KUKA KRL program: firepit2_1.src

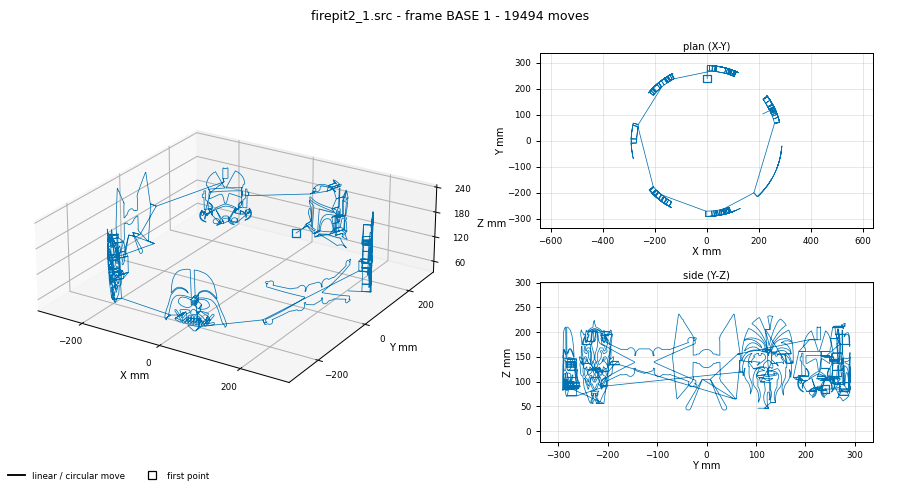
[picture p0: tool path of firepit2_1.src in frame BASE 1, 19494 of 19496 moves have a stored position in this frame; points joined in program order, loops and branches not executed]
&ACCESS RVP
&REL 1
&PARAM TEMPLATE = C:\KRC\Roboter\Template\vorgabe
&PARAM EDITMASK = *
DEF firepit2_1( )
EXT BAS (BAS_COMMAND :IN,REAL :IN )
DECL EKI_STATUS RET

INT INDX
FOR INDX=1 TO 6
	$ACC_AXIS[INDX]=50
	$VEL_AXIS[INDX]=20
ENDFOR

$VEL.ORI1=200
$VEL.ORI2=200
$ACC.ORI1=100
$ACC.ORI2=100

$VEL.CP = 0.1

$ACC.CP = 1

$IPO_MODE = #TCP
$APO.CDIS = 0.5
$ADVANCE = 5

$ACT_TOOL = 1
$TOOL=TOOL_DATA[1]
$ACT_BASE = 1
$BASE=BASE_DATA[1]

RET=EKI_Init("oxy")
RET=EKI_Open("oxy")

RET=EKI_SetBool("oxy","torchState",FALSE)
RET = EKI_Send("oxy","torchState")
PTP {A1 0.0,A2 -100.0,A3 150.0,A4 0.0,A5 -50.0,A6 0.0}

LIN {X 2.269,Y 239.989,Z 85.092,A -90.542,B 90.000,C 0.000} C_DIS
LIN {X 2.723,Y 287.987,Z 85.092,A -90.542,B 90.000,C 0.000} C_DIS
LIN {X 2.742,Y 289.987,Z 85.092,A -90.542,B 90.000,C 0.000} C_DIS
WAIT SEC 1
RET=EKI_SetBool("oxy","torchState",TRUE)
RET = EKI_Send("oxy","torchState")
LIN {X 3.106,Y 289.983,Z 85.575,A -90.614,B 90.000,C 0.000} C_DIS
LIN {X 4.946,Y 289.953,Z 87.268,A -90.977,B 90.000,C 0.000} C_DIS
LIN {X 6.840,Y 289.911,Z 88.899,A -91.352,B 90.000,C 0.000} C_DIS
LIN {X 8.695,Y 289.870,Z 90.495,A -91.718,B 90.000,C 0.000} C_DIS
LIN {X 10.282,Y 289.814,Z 88.565,A -92.032,B 90.000,C 0.000} C_DIS
LIN {X 11.858,Y 289.753,Z 86.625,A -92.343,B 90.000,C 0.000} C_DIS
LIN {X 13.089,Y 289.704,Z 85.109,A -92.587,B 90.000,C 0.000} C_DIS
LIN {X 13.703,Y 289.676,Z 84.499,A -92.708,B 90.000,C 0.000} C_DIS
LIN {X 13.987,Y 289.663,Z 84.366,A -92.764,B 90.000,C 0.000} C_DIS
LIN {X 14.006,Y 289.662,Z 86.866,A -92.768,B 90.000,C 0.000} C_DIS
LIN {X 14.025,Y 289.661,Z 89.365,A -92.772,B 90.000,C 0.000} C_DIS
LIN {X 14.045,Y 289.660,Z 91.865,A -92.776,B 90.000,C 0.000} C_DIS
LIN {X 14.064,Y 289.659,Z 94.365,A -92.780,B 90.000,C 0.000} C_DIS
LIN {X 14.084,Y 289.658,Z 96.865,A -92.784,B 90.000,C 0.000} C_DIS
LIN {X 14.103,Y 289.657,Z 99.365,A -92.788,B 90.000,C 0.000} C_DIS
LIN {X 14.116,Y 289.656,Z 101.865,A -92.790,B 90.000,C 0.000} C_DIS
LIN {X 14.110,Y 289.657,Z 104.365,A -92.789,B 90.000,C 0.000} C_DIS
LIN {X 14.104,Y 289.657,Z 106.864,A -92.788,B 90.000,C 0.000} C_DIS
LIN {X 14.098,Y 289.657,Z 109.364,A -92.786,B 90.000,C 0.000} C_DIS
LIN {X 14.092,Y 289.657,Z 111.864,A -92.785,B 90.000,C 0.000} C_DIS
LIN {X 14.086,Y 289.658,Z 114.364,A -92.784,B 90.000,C 0.000} C_DIS
LIN {X 14.080,Y 289.658,Z 116.864,A -92.783,B 90.000,C 0.000} C_DIS
LIN {X 14.074,Y 289.658,Z 119.364,A -92.782,B 90.000,C 0.000} C_DIS
LIN {X 13.921,Y 289.666,Z 121.859,A -92.751,B 90.000,C 0.000} C_DIS
LIN {X 13.726,Y 289.675,Z 124.352,A -92.713,B 90.000,C 0.000} C_DIS
LIN {X 13.394,Y 289.691,Z 126.829,A -92.647,B 90.000,C 0.000} C_DIS
LIN {X 12.905,Y 289.713,Z 129.281,A -92.550,B 90.000,C 0.000} C_DIS
LIN {X 12.266,Y 289.740,Z 131.697,A -92.424,B 90.000,C 0.000} C_DIS
LIN {X 11.477,Y 289.773,Z 134.069,A -92.268,B 90.000,C 0.000} C_DIS
LIN {X 10.547,Y 289.808,Z 136.390,A -92.084,B 90.000,C 0.000} C_DIS
LIN {X 9.438,Y 289.844,Z 138.630,A -91.865,B 90.000,C 0.000} C_DIS
LIN {X 8.303,Y 289.880,Z 140.857,A -91.641,B 90.000,C 0.000} C_DIS
LIN {X 7.391,Y 289.906,Z 142.534,A -91.460,B 90.000,C 0.000} C_DIS
LIN {X 7.419,Y 289.905,Z 145.034,A -91.466,B 90.000,C 0.000} C_DIS
LIN {X 7.484,Y 289.903,Z 147.533,A -91.479,B 90.000,C 0.000} C_DIS
LIN {X 7.552,Y 289.902,Z 149.639,A -91.492,B 90.000,C 0.000} C_DIS
LIN {X 7.695,Y 289.898,Z 150.255,A -91.521,B 90.000,C 0.000} C_DIS
LIN {X 7.879,Y 289.893,Z 150.291,A -91.557,B 90.000,C 0.000} C_DIS
LIN {X 8.002,Y 289.890,Z 150.193,A -91.581,B 90.000,C 0.000} C_DIS
LIN {X 8.394,Y 289.878,Z 148.728,A -91.659,B 90.000,C 0.000} C_DIS
LIN {X 8.824,Y 289.866,Z 147.667,A -91.744,B 90.000,C 0.000} C_DIS
LIN {X 9.375,Y 289.848,Z 146.647,A -91.853,B 90.000,C 0.000} C_DIS
LIN {X 10.028,Y 289.827,Z 145.711,A -91.982,B 90.000,C 0.000} C_DIS
LIN {X 11.083,Y 289.788,Z 144.578,A -92.190,B 90.000,C 0.000} C_DIS
LIN {X 13.041,Y 289.706,Z 143.026,A -92.577,B 90.000,C 0.000} C_DIS
LIN {X 15.151,Y 289.602,Z 141.689,A -92.995,B 90.000,C 0.000} C_DIS
LIN {X 17.324,Y 289.482,Z 140.459,A -93.425,B 90.000,C 0.000} C_DIS
LIN {X 17.924,Y 289.446,Z 140.050,A -93.544,B 90.000,C 0.000} C_DIS
LIN {X 18.369,Y 289.418,Z 139.616,A -93.632,B 90.000,C 0.000} C_DIS
LIN {X 18.808,Y 289.389,Z 139.037,A -93.719,B 90.000,C 0.000} C_DIS
LIN {X 19.190,Y 289.364,Z 138.387,A -93.794,B 90.000,C 0.000} C_DIS
LIN {X 19.466,Y 289.346,Z 137.743,A -93.849,B 90.000,C 0.000} C_DIS
LIN {X 19.578,Y 289.338,Z 137.136,A -93.871,B 90.000,C 0.000} C_DIS
LIN {X 19.405,Y 289.350,Z 134.642,A -93.837,B 90.000,C 0.000} C_DIS
LIN {X 19.241,Y 289.361,Z 132.148,A -93.804,B 90.000,C 0.000} C_DIS
LIN {X 19.076,Y 289.372,Z 129.653,A -93.772,B 90.000,C 0.000} C_DIS
LIN {X 18.917,Y 289.382,Z 127.158,A -93.740,B 90.000,C 0.000} C_DIS
LIN {X 18.761,Y 289.391,Z 124.663,A -93.709,B 90.000,C 0.000} C_DIS
LIN {X 18.606,Y 289.401,Z 122.168,A -93.678,B 90.000,C 0.000} C_DIS
LIN {X 18.450,Y 289.410,Z 119.673,A -93.648,B 90.000,C 0.000} C_DIS
LIN {X 18.294,Y 289.420,Z 117.178,A -93.617,B 90.000,C 0.000} C_DIS
LIN {X 18.138,Y 289.429,Z 114.683,A -93.586,B 90.000,C 0.000} C_DIS
LIN {X 17.983,Y 289.439,Z 112.188,A -93.555,B 90.000,C 0.000} C_DIS
LIN {X 17.827,Y 289.448,Z 109.693,A -93.524,B 90.000,C 0.000} C_DIS
LIN {X 17.671,Y 289.458,Z 107.198,A -93.493,B 90.000,C 0.000} C_DIS
LIN {X 17.515,Y 289.467,Z 104.703,A -93.463,B 90.000,C 0.000} C_DIS
LIN {X 17.359,Y 289.477,Z 102.208,A -93.432,B 90.000,C 0.000} C_DIS
LIN {X 17.204,Y 289.486,Z 99.713,A -93.401,B 90.000,C 0.000} C_DIS
LIN {X 17.048,Y 289.496,Z 97.218,A -93.370,B 90.000,C 0.000} C_DIS
LIN {X 16.892,Y 289.505,Z 94.723,A -93.339,B 90.000,C 0.000} C_DIS
LIN {X 16.736,Y 289.515,Z 92.228,A -93.308,B 90.000,C 0.000} C_DIS
LIN {X 16.580,Y 289.524,Z 89.733,A -93.278,B 90.000,C 0.000} C_DIS
LIN {X 16.425,Y 289.534,Z 87.238,A -93.247,B 90.000,C 0.000} C_DIS
LIN {X 16.269,Y 289.543,Z 84.743,A -93.216,B 90.000,C 0.000} C_DIS
LIN {X 16.179,Y 289.548,Z 83.458,A -93.198,B 90.000,C 0.000} C_DIS
LIN {X 18.542,Y 289.403,Z 82.655,A -93.666,B 90.000,C 0.000} C_DIS
LIN {X 20.897,Y 289.243,Z 81.832,A -94.132,B 90.000,C 0.000} C_DIS
LIN {X 23.250,Y 289.066,Z 81.005,A -94.598,B 90.000,C 0.000} C_DIS
LIN {X 24.631,Y 288.952,Z 80.507,A -94.872,B 90.000,C 0.000} C_DIS
LIN {X 23.274,Y 289.064,Z 78.411,A -94.603,B 90.000,C 0.000} C_DIS
LIN {X 21.895,Y 289.172,Z 76.398,A -94.330,B 90.000,C 0.000} C_DIS
LIN {X 19.621,Y 289.332,Z 77.424,A -93.880,B 90.000,C 0.000} C_DIS
LIN {X 17.348,Y 289.477,Z 78.455,A -93.430,B 90.000,C 0.000} C_DIS
LIN {X 15.074,Y 289.606,Z 79.486,A -92.980,B 90.000,C 0.000} C_DIS
LIN {X 12.800,Y 289.716,Z 80.517,A -92.530,B 90.000,C 0.000} C_DIS
LIN {X 10.524,Y 289.807,Z 81.548,A -92.080,B 90.000,C 0.000} C_DIS
LIN {X 8.248,Y 289.880,Z 82.580,A -91.630,B 90.000,C 0.000} C_DIS
LIN {X 5.972,Y 289.936,Z 83.611,A -91.180,B 90.000,C 0.000} C_DIS
LIN {X 3.698,Y 289.975,Z 84.650,A -90.731,B 90.000,C 0.000} C_DIS
LIN {X 2.742,Y 289.987,Z 85.092,A -90.542,B 90.000,C 0.000} C_DIS
LIN {X 2.723,Y 287.987,Z 85.092,A -90.542,B 90.000,C 0.000} C_DIS
WAIT SEC 0.1
RET=EKI_SetBool("oxy","torchState",FALSE)
RET = EKI_Send("oxy","torchState")
LIN {X 2.553,Y 269.988,Z 85.092,A -90.542,B 90.000,C 0.000} C_DIS
LIN {X 10.715,Y 269.787,Z 97.827,A -92.274,B 90.000,C 0.000} C_DIS
LIN {X 11.429,Y 287.773,Z 97.827,A -92.274,B 90.000,C 0.000} C_DIS
LIN {X 11.508,Y 289.772,Z 97.827,A -92.274,B 90.000,C 0.000} C_DIS
WAIT SEC 1
RET=EKI_SetBool("oxy","torchState",TRUE)
RET = EKI_Send("oxy","torchState")
LIN {X 11.733,Y 289.763,Z 98.367,A -92.319,B 90.000,C 0.000} C_DIS
LIN {X 12.293,Y 289.739,Z 100.803,A -92.430,B 90.000,C 0.000} C_DIS
LIN {X 12.626,Y 289.725,Z 103.281,A -92.495,B 90.000,C 0.000} C_DIS
LIN {X 12.812,Y 289.717,Z 105.774,A -92.532,B 90.000,C 0.000} C_DIS
LIN {X 12.854,Y 289.715,Z 108.274,A -92.540,B 90.000,C 0.000} C_DIS
LIN {X 12.814,Y 289.717,Z 110.773,A -92.533,B 90.000,C 0.000} C_DIS
LIN {X 12.625,Y 289.725,Z 113.266,A -92.495,B 90.000,C 0.000} C_DIS
LIN {X 12.426,Y 289.734,Z 115.758,A -92.456,B 90.000,C 0.000} C_DIS
LIN {X 12.102,Y 289.747,Z 118.237,A -92.392,B 90.000,C 0.000} C_DIS
LIN {X 11.760,Y 289.761,Z 120.713,A -92.324,B 90.000,C 0.000} C_DIS
LIN {X 11.291,Y 289.780,Z 123.169,A -92.231,B 90.000,C 0.000} C_DIS
LIN {X 10.772,Y 289.800,Z 125.614,A -92.129,B 90.000,C 0.000} C_DIS
LIN {X 10.082,Y 289.825,Z 128.017,A -91.992,B 90.000,C 0.000} C_DIS
LIN {X 9.685,Y 289.838,Z 128.998,A -91.914,B 90.000,C 0.000} C_DIS
LIN {X 9.310,Y 289.851,Z 129.580,A -91.840,B 90.000,C 0.000} C_DIS
LIN {X 8.906,Y 289.863,Z 129.935,A -91.760,B 90.000,C 0.000} C_DIS
LIN {X 8.480,Y 289.876,Z 130.055,A -91.676,B 90.000,C 0.000} C_DIS
LIN {X 8.053,Y 289.888,Z 129.956,A -91.591,B 90.000,C 0.000} C_DIS
LIN {X 7.635,Y 289.899,Z 129.594,A -91.509,B 90.000,C 0.000} C_DIS
LIN {X 7.309,Y 289.908,Z 129.126,A -91.444,B 90.000,C 0.000} C_DIS
LIN {X 6.981,Y 289.916,Z 128.453,A -91.379,B 90.000,C 0.000} C_DIS
LIN {X 6.222,Y 289.933,Z 126.072,A -91.229,B 90.000,C 0.000} C_DIS
LIN {X 5.689,Y 289.944,Z 123.629,A -91.124,B 90.000,C 0.000} C_DIS
LIN {X 5.315,Y 289.951,Z 121.157,A -91.050,B 90.000,C 0.000} C_DIS
LIN {X 5.080,Y 289.955,Z 118.668,A -91.004,B 90.000,C 0.000} C_DIS
LIN {X 4.862,Y 289.959,Z 116.354,A -90.961,B 90.000,C 0.000} C_DIS
LIN {X 4.950,Y 289.958,Z 115.800,A -90.978,B 90.000,C 0.000} C_DIS
LIN {X 6.205,Y 289.933,Z 113.638,A -91.226,B 90.000,C 0.000} C_DIS
LIN {X 6.480,Y 289.928,Z 113.155,A -91.280,B 90.000,C 0.000} C_DIS
LIN {X 7.462,Y 289.904,Z 110.856,A -91.474,B 90.000,C 0.000} C_DIS
LIN {X 8.309,Y 289.880,Z 108.504,A -91.642,B 90.000,C 0.000} C_DIS
LIN {X 9.087,Y 289.857,Z 106.128,A -91.796,B 90.000,C 0.000} C_DIS
LIN {X 9.799,Y 289.834,Z 103.732,A -91.936,B 90.000,C 0.000} C_DIS
LIN {X 10.498,Y 289.809,Z 101.332,A -92.075,B 90.000,C 0.000} C_DIS
LIN {X 11.191,Y 289.783,Z 98.930,A -92.211,B 90.000,C 0.000} C_DIS
LIN {X 11.508,Y 289.772,Z 97.827,A -92.274,B 90.000,C 0.000} C_DIS
LIN {X 11.429,Y 287.773,Z 97.827,A -92.274,B 90.000,C 0.000} C_DIS
WAIT SEC 0.1
RET=EKI_SetBool("oxy","torchState",FALSE)
RET = EKI_Send("oxy","torchState")
LIN {X 10.715,Y 269.787,Z 97.827,A -92.274,B 90.000,C 0.000} C_DIS
LIN {X 30.888,Y 268.227,Z 79.694,A -96.569,B 90.000,C 0.000} C_DIS
LIN {X 32.947,Y 286.109,Z 79.694,A -96.569,B 90.000,C 0.000} C_DIS
LIN {X 33.176,Y 288.096,Z 79.694,A -96.569,B 90.000,C 0.000} C_DIS
WAIT SEC 1
RET=EKI_SetBool("oxy","torchState",TRUE)
RET = EKI_Send("oxy","torchState")
LIN {X 31.366,Y 288.299,Z 79.726,A -96.209,B 90.000,C 0.000} C_DIS
LIN {X 31.245,Y 288.312,Z 79.795,A -96.185,B 90.000,C 0.000} C_DIS
LIN {X 31.374,Y 288.298,Z 82.291,A -96.211,B 90.000,C 0.000} C_DIS
LIN {X 31.521,Y 288.282,Z 84.787,A -96.240,B 90.000,C 0.000} C_DIS
LIN {X 31.668,Y 288.266,Z 87.283,A -96.269,B 90.000,C 0.000} C_DIS
LIN {X 31.819,Y 288.249,Z 89.778,A -96.299,B 90.000,C 0.000} C_DIS
LIN {X 31.971,Y 288.232,Z 92.273,A -96.329,B 90.000,C 0.000} C_DIS
LIN {X 32.123,Y 288.215,Z 94.768,A -96.360,B 90.000,C 0.000} C_DIS
LIN {X 32.275,Y 288.198,Z 97.264,A -96.390,B 90.000,C 0.000} C_DIS
LIN {X 32.427,Y 288.181,Z 99.759,A -96.420,B 90.000,C 0.000} C_DIS
LIN {X 32.579,Y 288.164,Z 102.254,A -96.450,B 90.000,C 0.000} C_DIS
LIN {X 32.731,Y 288.147,Z 104.749,A -96.481,B 90.000,C 0.000} C_DIS
LIN {X 32.878,Y 288.130,Z 107.245,A -96.510,B 90.000,C 0.000} C_DIS
LIN {X 33.024,Y 288.114,Z 109.741,A -96.539,B 90.000,C 0.000} C_DIS
LIN {X 33.165,Y 288.097,Z 112.236,A -96.567,B 90.000,C 0.000} C_DIS
LIN {X 33.305,Y 288.081,Z 114.732,A -96.595,B 90.000,C 0.000} C_DIS
LIN {X 33.446,Y 288.065,Z 117.228,A -96.623,B 90.000,C 0.000} C_DIS
LIN {X 33.590,Y 288.048,Z 119.724,A -96.651,B 90.000,C 0.000} C_DIS
LIN {X 33.747,Y 288.030,Z 122.219,A -96.683,B 90.000,C 0.000} C_DIS
LIN {X 33.904,Y 288.011,Z 124.714,A -96.714,B 90.000,C 0.000} C_DIS
LIN {X 34.055,Y 287.993,Z 127.209,A -96.744,B 90.000,C 0.000} C_DIS
LIN {X 34.202,Y 287.976,Z 129.705,A -96.773,B 90.000,C 0.000} C_DIS
LIN {X 34.346,Y 287.959,Z 132.200,A -96.802,B 90.000,C 0.000} C_DIS
LIN {X 34.409,Y 287.951,Z 133.346,A -96.814,B 90.000,C 0.000} C_DIS
LIN {X 34.518,Y 287.938,Z 133.760,A -96.836,B 90.000,C 0.000} C_DIS
LIN {X 34.705,Y 287.916,Z 134.075,A -96.873,B 90.000,C 0.000} C_DIS
LIN {X 34.992,Y 287.881,Z 134.376,A -96.930,B 90.000,C 0.000} C_DIS
LIN {X 35.373,Y 287.835,Z 134.609,A -97.006,B 90.000,C 0.000} C_DIS
LIN {X 36.438,Y 287.702,Z 134.880,A -97.218,B 90.000,C 0.000} C_DIS
LIN {X 38.916,Y 287.375,Z 134.943,A -97.712,B 90.000,C 0.000} C_DIS
LIN {X 41.391,Y 287.029,Z 134.988,A -98.206,B 90.000,C 0.000} C_DIS
LIN {X 43.863,Y 286.659,Z 135.032,A -98.700,B 90.000,C 0.000} C_DIS
LIN {X 46.332,Y 286.270,Z 135.076,A -99.193,B 90.000,C 0.000} C_DIS
LIN {X 48.798,Y 285.862,Z 135.148,A -99.687,B 90.000,C 0.000} C_DIS
LIN {X 51.256,Y 285.434,Z 135.304,A -100.180,B 90.000,C 0.000} C_DIS
LIN {X 53.709,Y 284.981,Z 135.460,A -100.673,B 90.000,C 0.000} C_DIS
LIN {X 56.159,Y 284.507,Z 135.616,A -101.166,B 90.000,C 0.000} C_DIS
LIN {X 58.601,Y 284.010,Z 135.814,A -101.658,B 90.000,C 0.000} C_DIS
LIN {X 61.038,Y 283.501,Z 136.040,A -102.150,B 90.000,C 0.000} C_DIS
LIN {X 63.463,Y 282.964,Z 136.326,A -102.641,B 90.000,C 0.000} C_DIS
LIN {X 65.880,Y 282.414,Z 136.644,A -103.131,B 90.000,C 0.000} C_DIS
LIN {X 68.285,Y 281.844,Z 137.022,A -103.619,B 90.000,C 0.000} C_DIS
LIN {X 70.670,Y 281.253,Z 137.484,A -104.105,B 90.000,C 0.000} C_DIS
LIN {X 73.034,Y 280.648,Z 138.026,A -104.587,B 90.000,C 0.000} C_DIS
LIN {X 75.378,Y 280.032,Z 138.640,A -105.066,B 90.000,C 0.000} C_DIS
LIN {X 76.863,Y 279.629,Z 139.139,A -105.370,B 90.000,C 0.000} C_DIS
LIN {X 76.918,Y 279.613,Z 139.927,A -105.381,B 90.000,C 0.000} C_DIS
LIN {X 76.873,Y 279.626,Z 140.646,A -105.372,B 90.000,C 0.000} C_DIS
LIN {X 74.460,Y 280.277,Z 140.616,A -104.878,B 90.000,C 0.000} C_DIS
LIN {X 72.040,Y 280.907,Z 140.607,A -104.384,B 90.000,C 0.000} C_DIS
LIN {X 69.616,Y 281.516,Z 140.598,A -103.890,B 90.000,C 0.000} C_DIS
LIN {X 67.186,Y 282.106,Z 140.611,A -103.396,B 90.000,C 0.000} C_DIS
LIN {X 64.753,Y 282.676,Z 140.646,A -102.902,B 90.000,C 0.000} C_DIS
LIN {X 62.314,Y 283.226,Z 140.681,A -102.408,B 90.000,C 0.000} C_DIS
LIN {X 59.872,Y 283.749,Z 140.789,A -101.915,B 90.000,C 0.000} C_DIS
LIN {X 57.426,Y 284.253,Z 140.900,A -101.421,B 90.000,C 0.000} C_DIS
LIN {X 54.977,Y 284.737,Z 141.035,A -100.928,B 90.000,C 0.000} C_DIS
LIN {X 52.526,Y 285.200,Z 141.195,A -100.435,B 90.000,C 0.000} C_DIS
LIN {X 50.071,Y 285.643,Z 141.363,A -99.942,B 90.000,C 0.000} C_DIS
LIN {X 47.616,Y 286.064,Z 141.575,A -99.450,B 90.000,C 0.000} C_DIS
LIN {X 45.157,Y 286.461,Z 141.787,A -98.958,B 90.000,C 0.000} C_DIS
LIN {X 42.699,Y 286.837,Z 142.045,A -98.467,B 90.000,C 0.000} C_DIS
LIN {X 40.238,Y 287.192,Z 142.311,A -97.976,B 90.000,C 0.000} C_DIS
LIN {X 37.779,Y 287.521,Z 142.611,A -97.485,B 90.000,C 0.000} C_DIS
LIN {X 35.320,Y 287.838,Z 142.936,A -96.996,B 90.000,C 0.000} C_DIS
LIN {X 32.867,Y 288.124,Z 143.323,A -96.508,B 90.000,C 0.000} C_DIS
LIN {X 30.417,Y 288.398,Z 143.738,A -96.021,B 90.000,C 0.000} C_DIS
LIN {X 27.978,Y 288.642,Z 144.228,A -95.536,B 90.000,C 0.000} C_DIS
LIN {X 25.548,Y 288.867,Z 144.773,A -95.054,B 90.000,C 0.000} C_DIS
LIN {X 23.128,Y 289.075,Z 145.363,A -94.574,B 90.000,C 0.000} C_DIS
LIN {X 20.731,Y 289.253,Z 146.048,A -94.099,B 90.000,C 0.000} C_DIS
LIN {X 18.356,Y 289.415,Z 146.813,A -93.629,B 90.000,C 0.000} C_DIS
LIN {X 16.021,Y 289.555,Z 147.694,A -93.167,B 90.000,C 0.000} C_DIS
LIN {X 14.146,Y 289.655,Z 148.532,A -92.796,B 90.000,C 0.000} C_DIS
LIN {X 12.056,Y 289.749,Z 149.750,A -92.383,B 90.000,C 0.000} C_DIS
LIN {X 10.680,Y 289.803,Z 150.791,A -92.110,B 90.000,C 0.000} C_DIS
LIN {X 9.525,Y 289.844,Z 151.907,A -91.882,B 90.000,C 0.000} C_DIS
LIN {X 8.647,Y 289.871,Z 153.037,A -91.709,B 90.000,C 0.000} C_DIS
LIN {X 8.100,Y 289.887,Z 154.122,A -91.601,B 90.000,C 0.000} C_DIS
LIN {X 7.966,Y 289.891,Z 154.614,A -91.574,B 90.000,C 0.000} C_DIS
LIN {X 7.936,Y 289.891,Z 155.165,A -91.568,B 90.000,C 0.000} C_DIS
LIN {X 8.018,Y 289.889,Z 156.091,A -91.584,B 90.000,C 0.000} C_DIS
LIN {X 8.873,Y 289.864,Z 158.440,A -91.753,B 90.000,C 0.000} C_DIS
LIN {X 9.052,Y 289.859,Z 158.884,A -91.789,B 90.000,C 0.000} C_DIS
LIN {X 11.147,Y 289.779,Z 157.522,A -92.203,B 90.000,C 0.000} C_DIS
LIN {X 13.204,Y 289.689,Z 156.104,A -92.610,B 90.000,C 0.000} C_DIS
LIN {X 15.264,Y 289.598,Z 154.691,A -93.017,B 90.000,C 0.000} C_DIS
LIN {X 17.393,Y 289.476,Z 153.386,A -93.438,B 90.000,C 0.000} C_DIS
LIN {X 19.610,Y 289.333,Z 152.240,A -93.877,B 90.000,C 0.000} C_DIS
LIN {X 21.892,Y 289.170,Z 151.232,A -94.329,B 90.000,C 0.000} C_DIS
LIN {X 24.232,Y 288.984,Z 150.371,A -94.793,B 90.000,C 0.000} C_DIS
LIN {X 26.612,Y 288.774,Z 149.635,A -95.265,B 90.000,C 0.000} C_DIS
LIN {X 29.022,Y 288.541,Z 149.013,A -95.744,B 90.000,C 0.000} C_DIS
LIN {X 31.454,Y 288.286,Z 148.495,A -96.227,B 90.000,C 0.000} C_DIS
LIN {X 33.902,Y 288.008,Z 148.069,A -96.713,B 90.000,C 0.000} C_DIS
LIN {X 36.360,Y 287.709,Z 147.727,A -97.203,B 90.000,C 0.000} C_DIS
LIN {X 38.825,Y 287.389,Z 147.457,A -97.694,B 90.000,C 0.000} C_DIS
LIN {X 41.293,Y 287.043,Z 147.270,A -98.186,B 90.000,C 0.000} C_DIS
LIN {X 43.763,Y 286.676,Z 147.143,A -98.680,B 90.000,C 0.000} C_DIS
LIN {X 46.230,Y 286.288,Z 147.033,A -99.173,B 90.000,C 0.000} C_DIS
LIN {X 48.694,Y 285.879,Z 146.923,A -99.666,B 90.000,C 0.000} C_DIS
LIN {X 51.155,Y 285.450,Z 146.840,A -100.160,B 90.000,C 0.000} C_DIS
LIN {X 53.614,Y 284.998,Z 146.795,A -100.654,B 90.000,C 0.000} C_DIS
LIN {X 56.068,Y 284.526,Z 146.750,A -101.148,B 90.000,C 0.000} C_DIS
LIN {X 58.519,Y 284.032,Z 146.727,A -101.642,B 90.000,C 0.000} C_DIS
LIN {X 60.965,Y 283.518,Z 146.769,A -102.136,B 90.000,C 0.000} C_DIS
LIN {X 63.406,Y 282.983,Z 146.811,A -102.629,B 90.000,C 0.000} C_DIS
LIN {X 65.843,Y 282.425,Z 146.853,A -103.123,B 90.000,C 0.000} C_DIS
LIN {X 68.274,Y 281.847,Z 146.940,A -103.617,B 90.000,C 0.000} C_DIS
LIN {X 70.699,Y 281.249,Z 147.031,A -104.110,B 90.000,C 0.000} C_DIS
LIN {X 73.119,Y 280.629,Z 147.122,A -104.604,B 90.000,C 0.000} C_DIS
LIN {X 75.532,Y 279.983,Z 147.233,A -105.097,B 90.000,C 0.000} C_DIS
LIN {X 77.942,Y 279.329,Z 147.350,A -105.591,B 90.000,C 0.000} C_DIS
LIN {X 80.341,Y 278.640,Z 147.491,A -106.084,B 90.000,C 0.000} C_DIS
LIN {X 82.738,Y 277.946,Z 147.637,A -106.577,B 90.000,C 0.000} C_DIS
LIN {X 83.639,Y 277.677,Z 147.701,A -106.763,B 90.000,C 0.000} C_DIS
LIN {X 84.426,Y 277.439,Z 147.637,A -106.925,B 90.000,C 0.000} C_DIS
LIN {X 85.212,Y 277.198,Z 146.852,A -107.088,B 90.000,C 0.000} C_DIS
LIN {X 85.569,Y 277.088,Z 146.663,A -107.161,B 90.000,C 0.000} C_DIS
LIN {X 85.692,Y 277.050,Z 146.577,A -107.187,B 90.000,C 0.000} C_DIS
LIN {X 85.754,Y 277.031,Z 146.399,A -107.200,B 90.000,C 0.000} C_DIS
LIN {X 85.652,Y 277.063,Z 143.901,A -107.179,B 90.000,C 0.000} C_DIS
LIN {X 85.533,Y 277.099,Z 141.404,A -107.154,B 90.000,C 0.000} C_DIS
LIN {X 85.455,Y 277.124,Z 138.906,A -107.138,B 90.000,C 0.000} C_DIS
LIN {X 85.383,Y 277.146,Z 136.407,A -107.123,B 90.000,C 0.000} C_DIS
LIN {X 85.314,Y 277.167,Z 133.908,A -107.109,B 90.000,C 0.000} C_DIS
LIN {X 85.248,Y 277.187,Z 131.409,A -107.095,B 90.000,C 0.000} C_DIS
LIN {X 85.166,Y 277.212,Z 128.911,A -107.078,B 90.000,C 0.000} C_DIS
LIN {X 85.080,Y 277.239,Z 126.412,A -107.060,B 90.000,C 0.000} C_DIS
LIN {X 84.986,Y 277.268,Z 123.914,A -107.041,B 90.000,C 0.000} C_DIS
LIN {X 84.904,Y 277.293,Z 121.416,A -107.024,B 90.000,C 0.000} C_DIS
LIN {X 84.828,Y 277.316,Z 118.917,A -107.008,B 90.000,C 0.000} C_DIS
LIN {X 84.756,Y 277.338,Z 116.418,A -106.993,B 90.000,C 0.000} C_DIS
LIN {X 84.678,Y 277.362,Z 113.920,A -106.977,B 90.000,C 0.000} C_DIS
LIN {X 84.595,Y 277.387,Z 111.421,A -106.960,B 90.000,C 0.000} C_DIS
LIN {X 84.513,Y 277.412,Z 108.923,A -106.943,B 90.000,C 0.000} C_DIS
LIN {X 84.431,Y 277.437,Z 106.425,A -106.926,B 90.000,C 0.000} C_DIS
LIN {X 84.352,Y 277.461,Z 103.926,A -106.910,B 90.000,C 0.000} C_DIS
LIN {X 84.259,Y 277.490,Z 101.428,A -106.891,B 90.000,C 0.000} C_DIS
LIN {X 84.162,Y 277.519,Z 98.930,A -106.871,B 90.000,C 0.000} C_DIS
LIN {X 84.095,Y 277.539,Z 96.431,A -106.857,B 90.000,C 0.000} C_DIS
LIN {X 84.031,Y 277.559,Z 93.932,A -106.844,B 90.000,C 0.000} C_DIS
LIN {X 84.008,Y 277.566,Z 93.174,A -106.839,B 90.000,C 0.000} C_DIS
LIN {X 83.913,Y 277.594,Z 92.829,A -106.819,B 90.000,C 0.000} C_DIS
LIN {X 83.739,Y 277.647,Z 92.621,A -106.784,B 90.000,C 0.000} C_DIS
LIN {X 81.633,Y 278.273,Z 91.430,A -106.349,B 90.000,C 0.000} C_DIS
LIN {X 81.536,Y 278.302,Z 91.383,A -106.329,B 90.000,C 0.000} C_DIS
LIN {X 81.573,Y 278.291,Z 93.883,A -106.337,B 90.000,C 0.000} C_DIS
LIN {X 81.610,Y 278.280,Z 96.382,A -106.345,B 90.000,C 0.000} C_DIS
LIN {X 81.647,Y 278.269,Z 98.882,A -106.352,B 90.000,C 0.000} C_DIS
LIN {X 81.683,Y 278.259,Z 101.382,A -106.360,B 90.000,C 0.000} C_DIS
LIN {X 81.726,Y 278.246,Z 103.881,A -106.368,B 90.000,C 0.000} C_DIS
LIN {X 81.770,Y 278.233,Z 106.381,A -106.378,B 90.000,C 0.000} C_DIS
LIN {X 81.814,Y 278.220,Z 108.880,A -106.387,B 90.000,C 0.000} C_DIS
LIN {X 81.858,Y 278.207,Z 111.380,A -106.396,B 90.000,C 0.000} C_DIS
LIN {X 81.903,Y 278.194,Z 113.879,A -106.405,B 90.000,C 0.000} C_DIS
LIN {X 81.947,Y 278.181,Z 116.379,A -106.414,B 90.000,C 0.000} C_DIS
LIN {X 81.987,Y 278.169,Z 118.878,A -106.422,B 90.000,C 0.000} C_DIS
LIN {X 82.025,Y 278.158,Z 121.378,A -106.430,B 90.000,C 0.000} C_DIS
LIN {X 82.063,Y 278.147,Z 123.877,A -106.438,B 90.000,C 0.000} C_DIS
LIN {X 82.105,Y 278.134,Z 126.377,A -106.447,B 90.000,C 0.000} C_DIS
LIN {X 82.119,Y 278.130,Z 128.877,A -106.449,B 90.000,C 0.000} C_DIS
LIN {X 82.056,Y 278.149,Z 130.204,A -106.436,B 90.000,C 0.000} C_DIS
LIN {X 81.775,Y 278.232,Z 130.973,A -106.378,B 90.000,C 0.000} C_DIS
LIN {X 81.315,Y 278.367,Z 131.602,A -106.284,B 90.000,C 0.000} C_DIS
LIN {X 80.724,Y 278.538,Z 132.042,A -106.162,B 90.000,C 0.000} C_DIS
LIN {X 80.050,Y 278.733,Z 132.243,A -106.024,B 90.000,C 0.000} C_DIS
LIN {X 77.654,Y 279.406,Z 132.000,A -105.532,B 90.000,C 0.000} C_DIS
LIN {X 75.264,Y 280.057,Z 131.669,A -105.042,B 90.000,C 0.000} C_DIS
LIN {X 72.870,Y 280.688,Z 131.321,A -104.553,B 90.000,C 0.000} C_DIS
LIN {X 70.480,Y 281.298,Z 130.915,A -104.066,B 90.000,C 0.000} C_DIS
LIN {X 68.094,Y 281.890,Z 130.460,A -103.580,B 90.000,C 0.000} C_DIS
LIN {X 65.716,Y 282.449,Z 129.931,A -103.098,B 90.000,C 0.000} C_DIS
LIN {X 63.344,Y 282.995,Z 129.358,A -102.617,B 90.000,C 0.000} C_DIS
LIN {X 60.991,Y 283.512,Z 128.692,A -102.141,B 90.000,C 0.000} C_DIS
LIN {X 58.675,Y 283.999,Z 127.886,A -101.673,B 90.000,C 0.000} C_DIS
LIN {X 56.409,Y 284.458,Z 126.935,A -101.216,B 90.000,C 0.000} C_DIS
LIN {X 54.210,Y 284.887,Z 125.825,A -100.774,B 90.000,C 0.000} C_DIS
LIN {X 52.122,Y 285.277,Z 124.507,A -100.354,B 90.000,C 0.000} C_DIS
LIN {X 50.180,Y 285.625,Z 122.972,A -99.964,B 90.000,C 0.000} C_DIS
LIN {X 48.375,Y 285.936,Z 121.271,A -99.602,B 90.000,C 0.000} C_DIS
LIN {X 46.695,Y 286.214,Z 119.440,A -99.266,B 90.000,C 0.000} C_DIS
LIN {X 46.031,Y 286.323,Z 118.709,A -99.133,B 90.000,C 0.000} C_DIS
LIN {X 44.565,Y 286.554,Z 116.698,A -98.840,B 90.000,C 0.000} C_DIS
LIN {X 43.228,Y 286.759,Z 114.595,A -98.573,B 90.000,C 0.000} C_DIS
LIN {X 42.019,Y 286.939,Z 112.415,A -98.331,B 90.000,C 0.000} C_DIS
LIN {X 40.925,Y 287.098,Z 110.172,A -98.113,B 90.000,C 0.000} C_DIS
LIN {X 40.001,Y 287.227,Z 107.853,A -97.928,B 90.000,C 0.000} C_DIS
LIN {X 39.171,Y 287.342,Z 105.498,A -97.763,B 90.000,C 0.000} C_DIS
LIN {X 38.415,Y 287.444,Z 103.117,A -97.612,B 90.000,C 0.000} C_DIS
LIN {X 37.801,Y 287.525,Z 100.695,A -97.490,B 90.000,C 0.000} C_DIS
LIN {X 37.242,Y 287.599,Z 98.259,A -97.378,B 90.000,C 0.000} C_DIS
LIN {X 36.760,Y 287.661,Z 95.807,A -97.282,B 90.000,C 0.000} C_DIS
LIN {X 36.360,Y 287.711,Z 93.340,A -97.203,B 90.000,C 0.000} C_DIS
LIN {X 35.997,Y 287.757,Z 90.867,A -97.130,B 90.000,C 0.000} C_DIS
LIN {X 35.724,Y 287.791,Z 88.382,A -97.076,B 90.000,C 0.000} C_DIS
LIN {X 35.466,Y 287.823,Z 85.896,A -97.025,B 90.000,C 0.000} C_DIS
LIN {X 35.288,Y 287.845,Z 83.402,A -96.989,B 90.000,C 0.000} C_DIS
LIN {X 35.119,Y 287.866,Z 80.908,A -96.956,B 90.000,C 0.000} C_DIS
LIN {X 35.084,Y 287.870,Z 80.148,A -96.949,B 90.000,C 0.000} C_DIS
LIN {X 33.176,Y 288.096,Z 79.694,A -96.569,B 90.000,C 0.000} C_DIS
LIN {X 32.947,Y 286.109,Z 79.694,A -96.569,B 90.000,C 0.000} C_DIS
WAIT SEC 0.1
RET=EKI_SetBool("oxy","torchState",FALSE)
RET = EKI_Send("oxy","torchState")
LIN {X 30.888,Y 268.227,Z 79.694,A -96.569,B 90.000,C 0.000} C_DIS
LIN {X 35.284,Y 267.685,Z 80.914,A -97.509,B 90.000,C 0.000} C_DIS
LIN {X 37.636,Y 285.530,Z 80.914,A -97.509,B 90.000,C 0.000} C_DIS
LIN {X 37.897,Y 287.513,Z 80.914,A -97.509,B 90.000,C 0.000} C_DIS
WAIT SEC 1
RET=EKI_SetBool("oxy","torchState",TRUE)
RET = EKI_Send("oxy","torchState")
LIN {X 37.966,Y 287.504,Z 80.893,A -97.523,B 90.000,C 0.000} C_DIS
LIN {X 40.414,Y 287.168,Z 81.272,A -98.011,B 90.000,C 0.000} C_DIS
LIN {X 42.855,Y 286.814,Z 81.680,A -98.498,B 90.000,C 0.000} C_DIS
LIN {X 45.291,Y 286.440,Z 82.098,A -98.985,B 90.000,C 0.000} C_DIS
LIN {X 47.715,Y 286.046,Z 82.565,A -99.470,B 90.000,C 0.000} C_DIS
LIN {X 50.135,Y 285.631,Z 83.039,A -99.955,B 90.000,C 0.000} C_DIS
LIN {X 52.538,Y 285.191,Z 83.569,A -100.438,B 90.000,C 0.000} C_DIS
LIN {X 54.939,Y 284.747,Z 84.106,A -100.920,B 90.000,C 0.000} C_DIS
LIN {X 57.319,Y 284.269,Z 84.703,A -101.400,B 90.000,C 0.000} C_DIS
LIN {X 59.695,Y 283.787,Z 85.310,A -101.879,B 90.000,C 0.000} C_DIS
LIN {X 62.050,Y 283.275,Z 85.976,A -102.355,B 90.000,C 0.000} C_DIS
LIN {X 64.398,Y 282.756,Z 86.659,A -102.830,B 90.000,C 0.000} C_DIS
LIN {X 66.724,Y 282.212,Z 87.397,A -103.302,B 90.000,C 0.000} C_DIS
LIN {X 69.039,Y 281.657,Z 88.160,A -103.773,B 90.000,C 0.000} C_DIS
LIN {X 71.333,Y 281.083,Z 88.971,A -104.240,B 90.000,C 0.000} C_DIS
LIN {X 73.611,Y 280.496,Z 89.817,A -104.705,B 90.000,C 0.000} C_DIS
LIN {X 75.870,Y 279.894,Z 90.701,A -105.167,B 90.000,C 0.000} C_DIS
LIN {X 77.563,Y 279.435,Z 91.401,A -105.513,B 90.000,C 0.000} C_DIS
LIN {X 77.805,Y 279.368,Z 91.576,A -105.563,B 90.000,C 0.000} C_DIS
LIN {X 77.358,Y 279.492,Z 94.033,A -105.471,B 90.000,C 0.000} C_DIS
LIN {X 76.827,Y 279.638,Z 96.471,A -105.362,B 90.000,C 0.000} C_DIS
LIN {X 76.254,Y 279.795,Z 98.900,A -105.245,B 90.000,C 0.000} C_DIS
LIN {X 75.580,Y 279.977,Z 101.300,A -105.107,B 90.000,C 0.000} C_DIS
LIN {X 74.887,Y 280.164,Z 103.695,A -104.965,B 90.000,C 0.000} C_DIS
LIN {X 74.080,Y 280.378,Z 106.051,A -104.800,B 90.000,C 0.000} C_DIS
LIN {X 73.239,Y 280.599,Z 108.395,A -104.628,B 90.000,C 0.000} C_DIS
LIN {X 72.279,Y 280.848,Z 110.690,A -104.432,B 90.000,C 0.000} C_DIS
LIN {X 71.196,Y 281.124,Z 112.926,A -104.212,B 90.000,C 0.000} C_DIS
LIN {X 69.936,Y 281.441,Z 115.061,A -103.955,B 90.000,C 0.000} C_DIS
LIN {X 69.719,Y 281.495,Z 115.408,A -103.911,B 90.000,C 0.000} C_DIS
LIN {X 68.618,Y 281.765,Z 116.792,A -103.687,B 90.000,C 0.000} C_DIS
LIN {X 67.561,Y 282.020,Z 117.728,A -103.472,B 90.000,C 0.000} C_DIS
LIN {X 66.938,Y 282.169,Z 118.106,A -103.345,B 90.000,C 0.000} C_DIS
LIN {X 66.346,Y 282.309,Z 118.348,A -103.225,B 90.000,C 0.000} C_DIS
LIN {X 65.711,Y 282.457,Z 118.476,A -103.096,B 90.000,C 0.000} C_DIS
LIN {X 63.275,Y 283.012,Z 118.374,A -102.603,B 90.000,C 0.000} C_DIS
LIN {X 60.866,Y 283.540,Z 117.969,A -102.115,B 90.000,C 0.000} C_DIS
LIN {X 58.490,Y 284.040,Z 117.373,A -101.636,B 90.000,C 0.000} C_DIS
LIN {X 56.181,Y 284.505,Z 116.535,A -101.170,B 90.000,C 0.000} C_DIS
LIN {X 53.973,Y 284.932,Z 115.444,A -100.726,B 90.000,C 0.000} C_DIS
LIN {X 51.890,Y 285.320,Z 114.118,A -100.307,B 90.000,C 0.000} C_DIS
LIN {X 49.979,Y 285.660,Z 112.542,A -99.924,B 90.000,C 0.000} C_DIS
LIN {X 48.229,Y 285.961,Z 110.783,A -99.573,B 90.000,C 0.000} C_DIS
LIN {X 46.658,Y 286.222,Z 108.856,A -99.259,B 90.000,C 0.000} C_DIS
LIN {X 45.273,Y 286.443,Z 106.786,A -98.982,B 90.000,C 0.000} C_DIS
LIN {X 43.992,Y 286.643,Z 104.649,A -98.725,B 90.000,C 0.000} C_DIS
LIN {X 42.849,Y 286.816,Z 102.432,A -98.497,B 90.000,C 0.000} C_DIS
LIN {X 41.823,Y 286.968,Z 100.157,A -98.292,B 90.000,C 0.000} C_DIS
LIN {X 40.965,Y 287.092,Z 97.813,A -98.121,B 90.000,C 0.000} C_DIS
LIN {X 40.272,Y 287.190,Z 95.413,A -97.982,B 90.000,C 0.000} C_DIS
LIN {X 39.691,Y 287.271,Z 92.983,A -97.867,B 90.000,C 0.000} C_DIS
LIN {X 39.205,Y 287.337,Z 90.531,A -97.770,B 90.000,C 0.000} C_DIS
LIN {X 38.738,Y 287.401,Z 88.076,A -97.677,B 90.000,C 0.000} C_DIS
LIN {X 38.383,Y 287.448,Z 85.602,A -97.606,B 90.000,C 0.000} C_DIS
LIN {X 38.077,Y 287.489,Z 83.121,A -97.545,B 90.000,C 0.000} C_DIS
LIN {X 37.873,Y 287.516,Z 81.055,A -97.504,B 90.000,C 0.000} C_DIS
LIN {X 37.897,Y 287.513,Z 80.914,A -97.509,B 90.000,C 0.000} C_DIS
LIN {X 37.636,Y 285.530,Z 80.914,A -97.509,B 90.000,C 0.000} C_DIS
WAIT SEC 0.1
RET=EKI_SetBool("oxy","torchState",FALSE)
RET = EKI_Send("oxy","torchState")
LIN {X 35.284,Y 267.685,Z 80.914,A -97.509,B 90.000,C 0.000} C_DIS
LIN {X 35.912,Y 267.601,Z 72.617,A -97.643,B 90.000,C 0.000} C_DIS
LIN {X 38.306,Y 285.441,Z 72.617,A -97.643,B 90.000,C 0.000} C_DIS
LIN {X 38.572,Y 287.423,Z 72.617,A -97.643,B 90.000,C 0.000} C_DIS
WAIT SEC 1
RET=EKI_SetBool("oxy","torchState",TRUE)
RET = EKI_Send("oxy","torchState")
LIN {X 40.990,Y 287.085,Z 73.157,A -98.126,B 90.000,C 0.000} C_DIS
LIN {X 43.374,Y 286.733,Z 73.822,A -98.602,B 90.000,C 0.000} C_DIS
LIN {X 45.725,Y 286.370,Z 74.590,A -99.072,B 90.000,C 0.000} C_DIS
LIN {X 48.036,Y 285.994,Z 75.467,A -99.534,B 90.000,C 0.000} C_DIS
LIN {X 50.342,Y 285.594,Z 76.344,A -99.997,B 90.000,C 0.000} C_DIS
LIN {X 52.641,Y 285.175,Z 77.233,A -100.459,B 90.000,C 0.000} C_DIS
LIN {X 54.936,Y 284.748,Z 78.127,A -100.920,B 90.000,C 0.000} C_DIS
LIN {X 55.997,Y 284.542,Z 78.456,A -101.133,B 90.000,C 0.000} C_DIS
LIN {X 56.759,Y 284.391,Z 78.584,A -101.287,B 90.000,C 0.000} C_DIS
LIN {X 59.204,Y 283.890,Z 78.723,A -101.780,B 90.000,C 0.000} C_DIS
LIN {X 61.645,Y 283.368,Z 78.861,A -102.273,B 90.000,C 0.000} C_DIS
LIN {X 64.082,Y 282.827,Z 79.000,A -102.766,B 90.000,C 0.000} C_DIS
LIN {X 66.514,Y 282.266,Z 79.138,A -103.259,B 90.000,C 0.000} C_DIS
LIN {X 68.942,Y 281.685,Z 79.276,A -103.753,B 90.000,C 0.000} C_DIS
LIN {X 71.363,Y 281.081,Z 79.413,A -104.246,B 90.000,C 0.000} C_DIS
LIN {X 73.780,Y 280.454,Z 79.551,A -104.739,B 90.000,C 0.000} C_DIS
LIN {X 76.191,Y 279.808,Z 79.689,A -105.232,B 90.000,C 0.000} C_DIS
LIN {X 78.595,Y 279.144,Z 79.859,A -105.725,B 90.000,C 0.000} C_DIS
LIN {X 80.989,Y 278.459,Z 80.075,A -106.217,B 90.000,C 0.000} C_DIS
LIN {X 83.378,Y 277.753,Z 80.291,A -106.709,B 90.000,C 0.000} C_DIS
LIN {X 85.757,Y 277.024,Z 80.535,A -107.201,B 90.000,C 0.000} C_DIS
LIN {X 88.123,Y 276.277,Z 80.836,A -107.691,B 90.000,C 0.000} C_DIS
LIN {X 90.482,Y 275.519,Z 81.173,A -108.180,B 90.000,C 0.000} C_DIS
LIN {X 92.822,Y 274.741,Z 81.582,A -108.668,B 90.000,C 0.000} C_DIS
LIN {X 95.128,Y 273.950,Z 82.137,A -109.149,B 90.000,C 0.000} C_DIS
LIN {X 96.079,Y 273.622,Z 82.383,A -109.348,B 90.000,C 0.000} C_DIS
LIN {X 98.295,Y 272.833,Z 83.229,A -109.813,B 90.000,C 0.000} C_DIS
LIN {X 99.204,Y 272.504,Z 83.577,A -110.004,B 90.000,C 0.000} C_DIS
LIN {X 100.686,Y 271.959,Z 81.639,A -110.316,B 90.000,C 0.000} C_DIS
LIN {X 102.219,Y 271.387,Z 79.748,A -110.639,B 90.000,C 0.000} C_DIS
LIN {X 103.834,Y 270.773,Z 77.941,A -110.980,B 90.000,C 0.000} C_DIS
LIN {X 105.533,Y 270.115,Z 76.230,A -111.340,B 90.000,C 0.000} C_DIS
LIN {X 107.316,Y 269.411,Z 74.625,A -111.719,B 90.000,C 0.000} C_DIS
LIN {X 109.180,Y 268.661,Z 73.137,A -112.116,B 90.000,C 0.000} C_DIS
LIN {X 111.119,Y 267.865,Z 71.775,A -112.530,B 90.000,C 0.000} C_DIS
LIN {X 113.125,Y 267.024,Z 70.543,A -112.960,B 90.000,C 0.000} C_DIS
LIN {X 115.195,Y 266.136,Z 69.459,A -113.405,B 90.000,C 0.000} C_DIS
LIN {X 117.308,Y 265.211,Z 68.495,A -113.861,B 90.000,C 0.000} C_DIS
LIN {X 119.450,Y 264.256,Z 67.630,A -114.324,B 90.000,C 0.000} C_DIS
LIN {X 120.727,Y 263.676,Z 67.108,A -114.601,B 90.000,C 0.000} C_DIS
LIN {X 120.930,Y 263.583,Z 66.971,A -114.645,B 90.000,C 0.000} C_DIS
LIN {X 120.982,Y 263.559,Z 66.851,A -114.657,B 90.000,C 0.000} C_DIS
LIN {X 120.789,Y 263.648,Z 66.808,A -114.615,B 90.000,C 0.000} C_DIS
LIN {X 118.600,Y 264.639,Z 67.498,A -114.140,B 90.000,C 0.000} C_DIS
LIN {X 116.407,Y 265.610,Z 68.205,A -113.666,B 90.000,C 0.000} C_DIS
LIN {X 114.151,Y 266.587,Z 68.660,A -113.180,B 90.000,C 0.000} C_DIS
LIN {X 111.856,Y 267.557,Z 68.861,A -112.688,B 90.000,C 0.000} C_DIS
LIN {X 109.546,Y 268.512,Z 68.852,A -112.194,B 90.000,C 0.000} C_DIS
LIN {X 107.237,Y 269.443,Z 68.626,A -111.702,B 90.000,C 0.000} C_DIS
LIN {X 104.954,Y 270.341,Z 68.143,A -111.218,B 90.000,C 0.000} C_DIS
LIN {X 102.715,Y 271.200,Z 67.436,A -110.744,B 90.000,C 0.000} C_DIS
LIN {X 100.515,Y 272.023,Z 66.582,A -110.280,B 90.000,C 0.000} C_DIS
LIN {X 98.354,Y 272.810,Z 65.601,A -109.825,B 90.000,C 0.000} C_DIS
LIN {X 96.234,Y 273.564,Z 64.512,A -109.381,B 90.000,C 0.000} C_DIS
LIN {X 94.159,Y 274.285,Z 63.318,A -108.947,B 90.000,C 0.000} C_DIS
LIN {X 92.100,Y 274.985,Z 62.085,A -108.517,B 90.000,C 0.000} C_DIS
LIN {X 91.174,Y 275.295,Z 61.543,A -108.324,B 90.000,C 0.000} C_DIS
LIN {X 90.478,Y 275.524,Z 61.253,A -108.179,B 90.000,C 0.000} C_DIS
LIN {X 89.860,Y 275.727,Z 61.091,A -108.051,B 90.000,C 0.000} C_DIS
LIN {X 88.836,Y 276.058,Z 61.069,A -107.838,B 90.000,C 0.000} C_DIS
LIN {X 86.959,Y 276.655,Z 61.763,A -107.449,B 90.000,C 0.000} C_DIS
LIN {X 84.607,Y 277.382,Z 62.199,A -106.963,B 90.000,C 0.000} C_DIS
LIN {X 82.252,Y 278.087,Z 62.651,A -106.477,B 90.000,C 0.000} C_DIS
LIN {X 79.896,Y 278.774,Z 63.127,A -105.992,B 90.000,C 0.000} C_DIS
LIN {X 77.534,Y 279.441,Z 63.603,A -105.507,B 90.000,C 0.000} C_DIS
LIN {X 75.167,Y 280.089,Z 64.078,A -105.022,B 90.000,C 0.000} C_DIS
LIN {X 72.793,Y 280.713,Z 64.554,A -104.537,B 90.000,C 0.000} C_DIS
LIN {X 70.414,Y 281.318,Z 65.027,A -104.052,B 90.000,C 0.000} C_DIS
LIN {X 68.030,Y 281.904,Z 65.499,A -103.567,B 90.000,C 0.000} C_DIS
LIN {X 65.641,Y 282.470,Z 65.972,A -103.082,B 90.000,C 0.000} C_DIS
LIN {X 63.248,Y 283.017,Z 66.444,A -102.597,B 90.000,C 0.000} C_DIS
LIN {X 60.850,Y 283.544,Z 66.916,A -102.112,B 90.000,C 0.000} C_DIS
LIN {X 58.448,Y 284.048,Z 67.388,A -101.627,B 90.000,C 0.000} C_DIS
LIN {X 56.041,Y 284.531,Z 67.861,A -101.142,B 90.000,C 0.000} C_DIS
LIN {X 53.628,Y 284.996,Z 68.319,A -100.657,B 90.000,C 0.000} C_DIS
LIN {X 51.209,Y 285.440,Z 68.772,A -100.171,B 90.000,C 0.000} C_DIS
LIN {X 48.788,Y 285.864,Z 69.224,A -99.685,B 90.000,C 0.000} C_DIS
LIN {X 46.362,Y 286.267,Z 69.677,A -99.199,B 90.000,C 0.000} C_DIS
LIN {X 43.934,Y 286.650,Z 70.129,A -98.714,B 90.000,C 0.000} C_DIS
LIN {X 41.501,Y 287.009,Z 70.578,A -98.228,B 90.000,C 0.000} C_DIS
LIN {X 39.064,Y 287.351,Z 71.022,A -97.742,B 90.000,C 0.000} C_DIS
LIN {X 36.619,Y 287.674,Z 71.428,A -97.254,B 90.000,C 0.000} C_DIS
LIN {X 34.169,Y 287.980,Z 71.817,A -96.766,B 90.000,C 0.000} C_DIS
LIN {X 34.136,Y 287.984,Z 71.823,A -96.760,B 90.000,C 0.000} C_DIS
LIN {X 34.060,Y 287.993,Z 71.904,A -96.745,B 90.000,C 0.000} C_DIS
LIN {X 34.090,Y 287.989,Z 72.022,A -96.751,B 90.000,C 0.000} C_DIS
LIN {X 34.338,Y 287.960,Z 72.156,A -96.800,B 90.000,C 0.000} C_DIS
LIN {X 36.812,Y 287.654,Z 72.351,A -97.293,B 90.000,C 0.000} C_DIS
LIN {X 38.572,Y 287.423,Z 72.617,A -97.643,B 90.000,C 0.000} C_DIS
LIN {X 38.306,Y 285.441,Z 72.617,A -97.643,B 90.000,C 0.000} C_DIS
WAIT SEC 0.1
RET=EKI_SetBool("oxy","torchState",FALSE)
RET = EKI_Send("oxy","torchState")
LIN {X 35.912,Y 267.601,Z 72.617,A -97.643,B 90.000,C 0.000} C_DIS
LIN {X 80.881,Y 257.601,Z 94.151,A -107.431,B 90.000,C 0.000} C_DIS
LIN {X 86.273,Y 274.774,Z 94.151,A -107.431,B 90.000,C 0.000} C_DIS
LIN {X 86.872,Y 276.682,Z 94.151,A -107.431,B 90.000,C 0.000} C_DIS
WAIT SEC 1
RET=EKI_SetBool("oxy","torchState",TRUE)
RET = EKI_Send("oxy","torchState")
LIN {X 86.997,Y 276.643,Z 96.648,A -107.457,B 90.000,C 0.000} C_DIS
LIN {X 87.130,Y 276.601,Z 99.144,A -107.485,B 90.000,C 0.000} C_DIS
LIN {X 87.263,Y 276.559,Z 101.640,A -107.512,B 90.000,C 0.000} C_DIS
LIN {X 87.396,Y 276.517,Z 104.136,A -107.540,B 90.000,C 0.000} C_DIS
LIN {X 87.526,Y 276.476,Z 106.632,A -107.567,B 90.000,C 0.000} C_DIS
LIN {X 87.653,Y 276.436,Z 109.128,A -107.593,B 90.000,C 0.000} C_DIS
LIN {X 87.781,Y 276.396,Z 111.625,A -107.619,B 90.000,C 0.000} C_DIS
LIN {X 87.908,Y 276.355,Z 114.121,A -107.646,B 90.000,C 0.000} C_DIS
LIN {X 88.047,Y 276.311,Z 116.616,A -107.675,B 90.000,C 0.000} C_DIS
LIN {X 88.051,Y 276.310,Z 116.669,A -107.675,B 90.000,C 0.000} C_DIS
LIN {X 90.333,Y 275.567,Z 117.369,A -108.150,B 90.000,C 0.000} C_DIS
LIN {X 92.623,Y 274.806,Z 118.021,A -108.626,B 90.000,C 0.000} C_DIS
LIN {X 94.921,Y 274.025,Z 118.622,A -109.106,B 90.000,C 0.000} C_DIS
LIN {X 95.004,Y 273.997,Z 118.643,A -109.123,B 90.000,C 0.000} C_DIS
LIN {X 94.930,Y 274.022,Z 116.145,A -109.108,B 90.000,C 0.000} C_DIS
LIN {X 94.857,Y 274.048,Z 113.646,A -109.092,B 90.000,C 0.000} C_DIS
LIN {X 94.783,Y 274.073,Z 111.147,A -109.077,B 90.000,C 0.000} C_DIS
LIN {X 94.709,Y 274.099,Z 108.649,A -109.061,B 90.000,C 0.000} C_DIS
LIN {X 94.635,Y 274.125,Z 106.150,A -109.046,B 90.000,C 0.000} C_DIS
LIN {X 94.561,Y 274.150,Z 103.651,A -109.031,B 90.000,C 0.000} C_DIS
LIN {X 94.492,Y 274.174,Z 101.152,A -109.016,B 90.000,C 0.000} C_DIS
LIN {X 94.482,Y 274.177,Z 100.805,A -109.014,B 90.000,C 0.000} C_DIS
LIN {X 94.176,Y 274.282,Z 100.351,A -108.950,B 90.000,C 0.000} C_DIS
LIN {X 92.361,Y 274.896,Z 98.745,A -108.572,B 90.000,C 0.000} C_DIS
LIN {X 90.529,Y 275.507,Z 97.158,A -108.190,B 90.000,C 0.000} C_DIS
LIN {X 88.696,Y 276.101,Z 95.566,A -107.809,B 90.000,C 0.000} C_DIS
LIN {X 87.164,Y 276.591,Z 94.209,A -107.492,B 90.000,C 0.000} C_DIS
LIN {X 86.956,Y 276.656,Z 94.088,A -107.449,B 90.000,C 0.000} C_DIS
LIN {X 86.872,Y 276.682,Z 94.151,A -107.431,B 90.000,C 0.000} C_DIS
LIN {X 86.273,Y 274.774,Z 94.151,A -107.431,B 90.000,C 0.000} C_DIS
WAIT SEC 0.1
RET=EKI_SetBool("oxy","torchState",FALSE)
RET = EKI_Send("oxy","torchState")
LIN {X 80.881,Y 257.601,Z 94.151,A -107.431,B 90.000,C 0.000} C_DIS
LIN {X 91.988,Y 253.847,Z 110.082,A -109.919,B 90.000,C 0.000} C_DIS
LIN {X 98.121,Y 270.770,Z 110.082,A -109.919,B 90.000,C 0.000} C_DIS
LIN {X 98.802,Y 272.650,Z 110.082,A -109.919,B 90.000,C 0.000} C_DIS
WAIT SEC 1
RET=EKI_SetBool("oxy","torchState",TRUE)
RET = EKI_Send("oxy","torchState")
LIN {X 98.993,Y 272.581,Z 110.094,A -109.960,B 90.000,C 0.000} C_DIS
LIN {X 99.494,Y 272.399,Z 110.195,A -110.065,B 90.000,C 0.000} C_DIS
LIN {X 101.837,Y 271.530,Z 110.240,A -110.559,B 90.000,C 0.000} C_DIS
LIN {X 104.172,Y 270.641,Z 110.132,A -111.052,B 90.000,C 0.000} C_DIS
LIN {X 106.498,Y 269.734,Z 110.007,A -111.545,B 90.000,C 0.000} C_DIS
LIN {X 108.816,Y 268.807,Z 109.883,A -112.039,B 90.000,C 0.000} C_DIS
LIN {X 110.911,Y 267.953,Z 109.734,A -112.486,B 90.000,C 0.000} C_DIS
LIN {X 111.087,Y 267.880,Z 112.227,A -112.523,B 90.000,C 0.000} C_DIS
LIN {X 111.252,Y 267.811,Z 114.720,A -112.559,B 90.000,C 0.000} C_DIS
LIN {X 111.402,Y 267.749,Z 117.215,A -112.591,B 90.000,C 0.000} C_DIS
LIN {X 111.523,Y 267.699,Z 119.711,A -112.617,B 90.000,C 0.000} C_DIS
LIN {X 111.644,Y 267.648,Z 122.208,A -112.642,B 90.000,C 0.000} C_DIS
LIN {X 111.764,Y 267.598,Z 124.704,A -112.668,B 90.000,C 0.000} C_DIS
LIN {X 111.885,Y 267.548,Z 127.201,A -112.694,B 90.000,C 0.000} C_DIS
LIN {X 112.005,Y 267.497,Z 129.697,A -112.720,B 90.000,C 0.000} C_DIS
LIN {X 112.162,Y 267.431,Z 132.191,A -112.753,B 90.000,C 0.000} C_DIS
LIN {X 112.208,Y 267.413,Z 133.419,A -112.763,B 90.000,C 0.000} C_DIS
LIN {X 112.045,Y 267.481,Z 134.228,A -112.728,B 90.000,C 0.000} C_DIS
LIN {X 111.791,Y 267.587,Z 134.621,A -112.674,B 90.000,C 0.000} C_DIS
LIN {X 111.408,Y 267.747,Z 134.953,A -112.592,B 90.000,C 0.000} C_DIS
LIN {X 110.909,Y 267.954,Z 135.220,A -112.485,B 90.000,C 0.000} C_DIS
LIN {X 110.308,Y 268.202,Z 135.420,A -112.357,B 90.000,C 0.000} C_DIS
LIN {X 108.853,Y 268.796,Z 135.602,A -112.046,B 90.000,C 0.000} C_DIS
LIN {X 107.149,Y 269.479,Z 135.470,A -111.683,B 90.000,C 0.000} C_DIS
LIN {X 105.816,Y 270.005,Z 135.095,A -111.400,B 90.000,C 0.000} C_DIS
LIN {X 105.295,Y 270.209,Z 134.820,A -111.290,B 90.000,C 0.000} C_DIS
LIN {X 104.886,Y 270.368,Z 134.495,A -111.203,B 90.000,C 0.000} C_DIS
LIN {X 104.610,Y 270.475,Z 134.161,A -111.145,B 90.000,C 0.000} C_DIS
LIN {X 104.400,Y 270.556,Z 133.720,A -111.100,B 90.000,C 0.000} C_DIS
LIN {X 103.825,Y 270.777,Z 131.297,A -110.979,B 90.000,C 0.000} C_DIS
LIN {X 103.258,Y 270.993,Z 128.872,A -110.859,B 90.000,C 0.000} C_DIS
LIN {X 102.689,Y 271.210,Z 126.448,A -110.738,B 90.000,C 0.000} C_DIS
LIN {X 102.108,Y 271.426,Z 124.026,A -110.616,B 90.000,C 0.000} C_DIS
LIN {X 101.526,Y 271.642,Z 121.604,A -110.493,B 90.000,C 0.000} C_DIS
LIN {X 100.945,Y 271.859,Z 119.182,A -110.371,B 90.000,C 0.000} C_DIS
LIN {X 100.363,Y 272.075,Z 116.761,A -110.248,B 90.000,C 0.000} C_DIS
LIN {X 99.782,Y 272.291,Z 114.339,A -110.126,B 90.000,C 0.000} C_DIS
LIN {X 99.204,Y 272.504,Z 111.916,A -110.004,B 90.000,C 0.000} C_DIS
LIN {X 98.791,Y 272.654,Z 110.167,A -109.917,B 90.000,C 0.000} C_DIS
LIN {X 98.802,Y 272.650,Z 110.082,A -109.919,B 90.000,C 0.000} C_DIS
LIN {X 98.121,Y 270.770,Z 110.082,A -109.919,B 90.000,C 0.000} C_DIS
WAIT SEC 0.1
RET=EKI_SetBool("oxy","torchState",FALSE)
RET = EKI_Send("oxy","torchState")
LIN {X 91.988,Y 253.847,Z 110.082,A -109.919,B 90.000,C 0.000} C_DIS
LIN {X 99.194,Y 251.119,Z 105.756,A -111.554,B 90.000,C 0.000} C_DIS
LIN {X 105.807,Y 267.860,Z 105.756,A -111.554,B 90.000,C 0.000} C_DIS
LIN {X 106.542,Y 269.720,Z 105.756,A -111.554,B 90.000,C 0.000} C_DIS
WAIT SEC 1
RET=EKI_SetBool("oxy","torchState",TRUE)
RET = EKI_Send("oxy","torchState")
LIN {X 106.840,Y 269.602,Z 106.290,A -111.618,B 90.000,C 0.000} C_DIS
LIN {X 107.270,Y 269.431,Z 106.746,A -111.709,B 90.000,C 0.000} C_DIS
LIN {X 107.820,Y 269.211,Z 107.109,A -111.826,B 90.000,C 0.000} C_DIS
LIN {X 108.708,Y 268.854,Z 107.454,A -112.015,B 90.000,C 0.000} C_DIS
LIN {X 109.735,Y 268.437,Z 107.538,A -112.234,B 90.000,C 0.000} C_DIS
LIN {X 112.034,Y 267.484,Z 107.303,A -112.726,B 90.000,C 0.000} C_DIS
LIN {X 114.295,Y 266.525,Z 106.839,A -113.211,B 90.000,C 0.000} C_DIS
LIN {X 116.544,Y 265.549,Z 106.348,A -113.696,B 90.000,C 0.000} C_DIS
LIN {X 118.780,Y 264.556,Z 105.835,A -114.179,B 90.000,C 0.000} C_DIS
LIN {X 119.766,Y 264.114,Z 105.581,A -114.393,B 90.000,C 0.000} C_DIS
LIN {X 118.103,Y 264.861,Z 103.870,A -114.032,B 90.000,C 0.000} C_DIS
LIN {X 116.706,Y 265.480,Z 102.532,A -113.731,B 90.000,C 0.000} C_DIS
LIN {X 116.682,Y 265.491,Z 102.127,A -113.725,B 90.000,C 0.000} C_DIS
LIN {X 117.071,Y 265.319,Z 99.663,A -113.809,B 90.000,C 0.000} C_DIS
LIN {X 117.091,Y 265.310,Z 99.535,A -113.814,B 90.000,C 0.000} C_DIS
LIN {X 117.064,Y 265.323,Z 99.436,A -113.808,B 90.000,C 0.000} C_DIS
LIN {X 115.122,Y 266.170,Z 100.763,A -113.389,B 90.000,C 0.000} C_DIS
LIN {X 113.057,Y 267.054,Z 101.860,A -112.945,B 90.000,C 0.000} C_DIS
LIN {X 112.173,Y 267.427,Z 102.234,A -112.756,B 90.000,C 0.000} C_DIS
LIN {X 110.761,Y 268.015,Z 102.645,A -112.453,B 90.000,C 0.000} C_DIS
LIN {X 108.466,Y 268.951,Z 102.975,A -111.964,B 90.000,C 0.000} C_DIS
LIN {X 108.018,Y 269.132,Z 103.038,A -111.868,B 90.000,C 0.000} C_DIS
LIN {X 107.290,Y 269.423,Z 103.277,A -111.713,B 90.000,C 0.000} C_DIS
LIN {X 106.829,Y 269.606,Z 103.594,A -111.615,B 90.000,C 0.000} C_DIS
LIN {X 106.524,Y 269.727,Z 104.013,A -111.551,B 90.000,C 0.000} C_DIS
LIN {X 106.376,Y 269.785,Z 104.535,A -111.519,B 90.000,C 0.000} C_DIS
LIN {X 106.386,Y 269.782,Z 105.160,A -111.521,B 90.000,C 0.000} C_DIS
LIN {X 106.542,Y 269.720,Z 105.756,A -111.554,B 90.000,C 0.000} C_DIS
LIN {X 105.807,Y 267.860,Z 105.756,A -111.554,B 90.000,C 0.000} C_DIS
WAIT SEC 0.1
RET=EKI_SetBool("oxy","torchState",FALSE)
RET = EKI_Send("oxy","torchState")
LIN {X 99.194,Y 251.119,Z 105.756,A -111.554,B 90.000,C 0.000} C_DIS
LIN {X 105.223,Y 248.652,Z 109.467,A -112.937,B 90.000,C 0.000} C_DIS
LIN {X 112.238,Y 265.229,Z 109.467,A -112.937,B 90.000,C 0.000} C_DIS
LIN {X 113.018,Y 267.071,Z 109.467,A -112.937,B 90.000,C 0.000} C_DIS
WAIT SEC 1
RET=EKI_SetBool("oxy","torchState",TRUE)
RET = EKI_Send("oxy","torchState")
LIN {X 115.290,Y 266.090,Z 109.119,A -113.426,B 90.000,C 0.000} C_DIS
LIN {X 117.558,Y 265.103,Z 108.749,A -113.914,B 90.000,C 0.000} C_DIS
LIN {X 119.792,Y 264.096,Z 108.256,A -114.399,B 90.000,C 0.000} C_DIS
LIN {X 121.740,Y 263.210,Z 107.800,A -114.822,B 90.000,C 0.000} C_DIS
LIN {X 121.478,Y 263.331,Z 110.283,A -114.765,B 90.000,C 0.000} C_DIS
LIN {X 121.182,Y 263.467,Z 112.761,A -114.700,B 90.000,C 0.000} C_DIS
LIN {X 120.885,Y 263.603,Z 115.240,A -114.636,B 90.000,C 0.000} C_DIS
LIN {X 120.590,Y 263.738,Z 117.719,A -114.571,B 90.000,C 0.000} C_DIS
LIN {X 120.297,Y 263.872,Z 120.198,A -114.508,B 90.000,C 0.000} C_DIS
LIN {X 120.004,Y 264.006,Z 122.677,A -114.444,B 90.000,C 0.000} C_DIS
LIN {X 119.716,Y 264.137,Z 125.157,A -114.382,B 90.000,C 0.000} C_DIS
LIN {X 119.375,Y 264.291,Z 127.628,A -114.308,B 90.000,C 0.000} C_DIS
LIN {X 118.856,Y 264.525,Z 129.934,A -114.195,B 90.000,C 0.000} C_DIS
LIN {X 118.362,Y 264.746,Z 131.184,A -114.088,B 90.000,C 0.000} C_DIS
LIN {X 118.014,Y 264.901,Z 131.810,A -114.013,B 90.000,C 0.000} C_DIS
LIN {X 117.599,Y 265.086,Z 132.372,A -113.923,B 90.000,C 0.000} C_DIS
LIN {X 117.150,Y 265.285,Z 132.831,A -113.826,B 90.000,C 0.000} C_DIS
LIN {X 116.701,Y 265.482,Z 133.147,A -113.729,B 90.000,C 0.000} C_DIS
LIN {X 116.233,Y 265.687,Z 133.337,A -113.628,B 90.000,C 0.000} C_DIS
LIN {X 115.733,Y 265.906,Z 133.441,A -113.521,B 90.000,C 0.000} C_DIS
LIN {X 115.249,Y 266.116,Z 133.454,A -113.416,B 90.000,C 0.000} C_DIS
LIN {X 114.835,Y 266.295,Z 133.370,A -113.327,B 90.000,C 0.000} C_DIS
LIN {X 114.416,Y 266.475,Z 133.066,A -113.237,B 90.000,C 0.000} C_DIS
LIN {X 114.222,Y 266.558,Z 132.674,A -113.195,B 90.000,C 0.000} C_DIS
LIN {X 114.090,Y 266.614,Z 130.178,A -113.167,B 90.000,C 0.000} C_DIS
LIN {X 113.958,Y 266.671,Z 127.682,A -113.139,B 90.000,C 0.000} C_DIS
LIN {X 113.827,Y 266.727,Z 125.187,A -113.111,B 90.000,C 0.000} C_DIS
LIN {X 113.695,Y 266.783,Z 122.691,A -113.082,B 90.000,C 0.000} C_DIS
LIN {X 113.564,Y 266.839,Z 120.195,A -113.054,B 90.000,C 0.000} C_DIS
LIN {X 113.432,Y 266.895,Z 117.699,A -113.026,B 90.000,C 0.000} C_DIS
LIN {X 113.300,Y 266.951,Z 115.203,A -112.998,B 90.000,C 0.000} C_DIS
LIN {X 113.169,Y 267.007,Z 112.708,A -112.969,B 90.000,C 0.000} C_DIS
LIN {X 113.040,Y 267.062,Z 110.212,A -112.942,B 90.000,C 0.000} C_DIS
LIN {X 113.018,Y 267.071,Z 109.467,A -112.937,B 90.000,C 0.000} C_DIS
LIN {X 112.238,Y 265.229,Z 109.467,A -112.937,B 90.000,C 0.000} C_DIS
WAIT SEC 0.1
RET=EKI_SetBool("oxy","torchState",FALSE)
RET = EKI_Send("oxy","torchState")
LIN {X 105.223,Y 248.652,Z 109.467,A -112.937,B 90.000,C 0.000} C_DIS
LIN {X 99.000,Y 251.195,Z 97.294,A -111.510,B 90.000,C 0.000} C_DIS
LIN {X 105.600,Y 267.942,Z 97.294,A -111.510,B 90.000,C 0.000} C_DIS
LIN {X 106.333,Y 269.802,Z 97.294,A -111.510,B 90.000,C 0.000} C_DIS
WAIT SEC 1
RET=EKI_SetBool("oxy","torchState",TRUE)
RET = EKI_Send("oxy","torchState")
LIN {X 106.205,Y 269.853,Z 97.444,A -111.483,B 90.000,C 0.000} C_DIS
LIN {X 108.525,Y 268.924,Z 97.408,A -111.977,B 90.000,C 0.000} C_DIS
LIN {X 110.839,Y 267.980,Z 97.325,A -112.470,B 90.000,C 0.000} C_DIS
LIN {X 113.144,Y 267.017,Z 97.241,A -112.964,B 90.000,C 0.000} C_DIS
LIN {X 115.435,Y 266.033,Z 97.056,A -113.457,B 90.000,C 0.000} C_DIS
LIN {X 115.899,Y 265.833,Z 97.019,A -113.556,B 90.000,C 0.000} C_DIS
LIN {X 116.509,Y 265.567,Z 96.864,A -113.688,B 90.000,C 0.000} C_DIS
LIN {X 116.961,Y 265.368,Z 96.621,A -113.786,B 90.000,C 0.000} C_DIS
LIN {X 117.518,Y 265.122,Z 96.134,A -113.906,B 90.000,C 0.000} C_DIS
LIN {X 117.792,Y 265.000,Z 95.692,A -113.965,B 90.000,C 0.000} C_DIS
LIN {X 118.153,Y 264.839,Z 94.336,A -114.043,B 90.000,C 0.000} C_DIS
LIN {X 118.339,Y 264.756,Z 93.996,A -114.083,B 90.000,C 0.000} C_DIS
LIN {X 120.007,Y 264.003,Z 92.293,A -114.445,B 90.000,C 0.000} C_DIS
LIN {X 121.707,Y 263.222,Z 90.635,A -114.815,B 90.000,C 0.000} C_DIS
LIN {X 123.253,Y 262.505,Z 89.086,A -115.151,B 90.000,C 0.000} C_DIS
LIN {X 121.370,Y 263.380,Z 88.625,A -114.741,B 90.000,C 0.000} C_DIS
LIN {X 119.108,Y 264.406,Z 88.344,A -114.250,B 90.000,C 0.000} C_DIS
LIN {X 118.184,Y 264.826,Z 88.229,A -114.050,B 90.000,C 0.000} C_DIS
LIN {X 115.895,Y 265.831,Z 88.208,A -113.556,B 90.000,C 0.000} C_DIS
LIN {X 113.599,Y 266.819,Z 88.237,A -113.062,B 90.000,C 0.000} C_DIS
LIN {X 111.298,Y 267.790,Z 88.352,A -112.569,B 90.000,C 0.000} C_DIS
LIN {X 108.999,Y 268.735,Z 88.622,A -112.077,B 90.000,C 0.000} C_DIS
LIN {X 106.708,Y 269.654,Z 89.019,A -111.590,B 90.000,C 0.000} C_DIS
LIN {X 105.607,Y 270.087,Z 89.285,A -111.356,B 90.000,C 0.000} C_DIS
LIN {X 105.034,Y 270.311,Z 89.590,A -111.235,B 90.000,C 0.000} C_DIS
LIN {X 104.842,Y 270.385,Z 89.753,A -111.194,B 90.000,C 0.000} C_DIS
LIN {X 107.131,Y 269.485,Z 90.198,A -111.680,B 90.000,C 0.000} C_DIS
LIN {X 108.000,Y 269.140,Z 90.385,A -111.864,B 90.000,C 0.000} C_DIS
LIN {X 108.562,Y 268.913,Z 90.613,A -111.984,B 90.000,C 0.000} C_DIS
LIN {X 109.020,Y 268.728,Z 90.903,A -112.082,B 90.000,C 0.000} C_DIS
LIN {X 109.471,Y 268.544,Z 91.370,A -112.178,B 90.000,C 0.000} C_DIS
LIN {X 109.708,Y 268.448,Z 91.787,A -112.229,B 90.000,C 0.000} C_DIS
LIN {X 109.481,Y 268.540,Z 92.127,A -112.180,B 90.000,C 0.000} C_DIS
LIN {X 109.056,Y 268.713,Z 92.496,A -112.090,B 90.000,C 0.000} C_DIS
LIN {X 107.897,Y 269.181,Z 92.903,A -111.843,B 90.000,C 0.000} C_DIS
LIN {X 107.879,Y 269.188,Z 93.016,A -111.839,B 90.000,C 0.000} C_DIS
LIN {X 108.458,Y 268.955,Z 93.632,A -111.962,B 90.000,C 0.000} C_DIS
LIN {X 108.486,Y 268.944,Z 93.850,A -111.968,B 90.000,C 0.000} C_DIS
LIN {X 108.418,Y 268.971,Z 94.084,A -111.954,B 90.000,C 0.000} C_DIS
LIN {X 108.072,Y 269.111,Z 94.375,A -111.880,B 90.000,C 0.000} C_DIS
LIN {X 106.527,Y 269.726,Z 94.811,A -111.551,B 90.000,C 0.000} C_DIS
LIN {X 106.302,Y 269.814,Z 94.970,A -111.504,B 90.000,C 0.000} C_DIS
LIN {X 107.526,Y 269.329,Z 95.396,A -111.764,B 90.000,C 0.000} C_DIS
LIN {X 107.712,Y 269.255,Z 95.555,A -111.803,B 90.000,C 0.000} C_DIS
LIN {X 107.803,Y 269.218,Z 95.768,A -111.823,B 90.000,C 0.000} C_DIS
LIN {X 107.798,Y 269.220,Z 96.170,A -111.821,B 90.000,C 0.000} C_DIS
LIN {X 107.589,Y 269.304,Z 96.505,A -111.777,B 90.000,C 0.000} C_DIS
LIN {X 106.333,Y 269.802,Z 97.294,A -111.510,B 90.000,C 0.000} C_DIS
LIN {X 105.600,Y 267.942,Z 97.294,A -111.510,B 90.000,C 0.000} C_DIS
WAIT SEC 0.1
RET=EKI_SetBool("oxy","torchState",FALSE)
RET = EKI_Send("oxy","torchState")
LIN {X 99.000,Y 251.195,Z 97.294,A -111.510,B 90.000,C 0.000} C_DIS
LIN {X 90.305,Y 254.450,Z 123.011,A -109.540,B 90.000,C 0.000} C_DIS
LIN {X 96.325,Y 271.414,Z 123.011,A -109.540,B 90.000,C 0.000} C_DIS
LIN {X 96.994,Y 273.299,Z 123.011,A -109.540,B 90.000,C 0.000} C_DIS
WAIT SEC 1
RET=EKI_SetBool("oxy","torchState",TRUE)
RET = EKI_Send("oxy","torchState")
LIN {X 97.071,Y 273.271,Z 125.509,A -109.556,B 90.000,C 0.000} C_DIS
LIN {X 97.142,Y 273.246,Z 128.008,A -109.571,B 90.000,C 0.000} C_DIS
LIN {X 97.214,Y 273.221,Z 130.507,A -109.586,B 90.000,C 0.000} C_DIS
LIN {X 97.315,Y 273.184,Z 133.004,A -109.607,B 90.000,C 0.000} C_DIS
LIN {X 97.344,Y 273.174,Z 133.505,A -109.613,B 90.000,C 0.000} C_DIS
LIN {X 99.066,Y 272.554,Z 134.171,A -109.975,B 90.000,C 0.000} C_DIS
LIN {X 99.066,Y 272.554,Z 135.418,A -109.975,B 90.000,C 0.000} C_DIS
LIN {X 98.745,Y 272.671,Z 135.529,A -109.907,B 90.000,C 0.000} C_DIS
LIN {X 97.809,Y 273.008,Z 135.641,A -109.711,B 90.000,C 0.000} C_DIS
LIN {X 96.966,Y 273.309,Z 135.568,A -109.534,B 90.000,C 0.000} C_DIS
LIN {X 94.702,Y 274.097,Z 134.857,A -109.060,B 90.000,C 0.000} C_DIS
LIN {X 92.439,Y 274.868,Z 134.127,A -108.588,B 90.000,C 0.000} C_DIS
LIN {X 90.171,Y 275.625,Z 133.399,A -108.115,B 90.000,C 0.000} C_DIS
LIN {X 89.463,Y 275.856,Z 133.163,A -107.968,B 90.000,C 0.000} C_DIS
LIN {X 89.463,Y 275.856,Z 130.906,A -107.968,B 90.000,C 0.000} C_DIS
LIN {X 90.283,Y 275.589,Z 131.156,A -108.139,B 90.000,C 0.000} C_DIS
LIN {X 90.387,Y 275.554,Z 131.084,A -108.160,B 90.000,C 0.000} C_DIS
LIN {X 90.733,Y 275.441,Z 128.611,A -108.232,B 90.000,C 0.000} C_DIS
LIN {X 91.022,Y 275.345,Z 126.510,A -108.293,B 90.000,C 0.000} C_DIS
LIN {X 93.384,Y 274.553,Z 126.724,A -108.785,B 90.000,C 0.000} C_DIS
LIN {X 94.099,Y 274.309,Z 126.782,A -108.934,B 90.000,C 0.000} C_DIS
LIN {X 94.503,Y 274.170,Z 126.626,A -109.018,B 90.000,C 0.000} C_DIS
LIN {X 95.274,Y 273.903,Z 125.461,A -109.180,B 90.000,C 0.000} C_DIS
LIN {X 93.059,Y 274.662,Z 124.583,A -108.717,B 90.000,C 0.000} C_DIS
LIN {X 90.839,Y 275.403,Z 123.705,A -108.255,B 90.000,C 0.000} C_DIS
LIN {X 90.288,Y 275.587,Z 123.487,A -108.140,B 90.000,C 0.000} C_DIS
LIN {X 90.071,Y 275.658,Z 123.470,A -108.095,B 90.000,C 0.000} C_DIS
LIN {X 90.040,Y 275.668,Z 125.969,A -108.088,B 90.000,C 0.000} C_DIS
LIN {X 90.045,Y 275.666,Z 127.429,A -108.089,B 90.000,C 0.000} C_DIS
LIN {X 89.903,Y 275.713,Z 127.429,A -108.060,B 90.000,C 0.000} C_DIS
LIN {X 88.604,Y 276.133,Z 127.194,A -107.790,B 90.000,C 0.000} C_DIS
LIN {X 88.366,Y 276.209,Z 127.109,A -107.741,B 90.000,C 0.000} C_DIS
LIN {X 88.266,Y 276.241,Z 126.987,A -107.720,B 90.000,C 0.000} C_DIS
LIN {X 88.229,Y 276.253,Z 124.488,A -107.712,B 90.000,C 0.000} C_DIS
LIN {X 88.225,Y 276.254,Z 121.988,A -107.712,B 90.000,C 0.000} C_DIS
LIN {X 88.231,Y 276.252,Z 120.903,A -107.713,B 90.000,C 0.000} C_DIS
LIN {X 88.312,Y 276.226,Z 120.434,A -107.729,B 90.000,C 0.000} C_DIS
LIN {X 90.604,Y 275.474,Z 121.088,A -108.206,B 90.000,C 0.000} C_DIS
LIN {X 92.887,Y 274.718,Z 121.771,A -108.681,B 90.000,C 0.000} C_DIS
LIN {X 95.161,Y 273.936,Z 122.456,A -109.156,B 90.000,C 0.000} C_DIS
LIN {X 96.994,Y 273.299,Z 123.011,A -109.540,B 90.000,C 0.000} C_DIS
LIN {X 96.325,Y 271.414,Z 123.011,A -109.540,B 90.000,C 0.000} C_DIS
WAIT SEC 0.1
RET=EKI_SetBool("oxy","torchState",FALSE)
RET = EKI_Send("oxy","torchState")
LIN {X 90.305,Y 254.450,Z 123.011,A -109.540,B 90.000,C 0.000} C_DIS
LIN {X 86.043,Y 255.923,Z 137.642,A -108.583,B 90.000,C 0.000} C_DIS
LIN {X 91.779,Y 272.985,Z 137.642,A -108.583,B 90.000,C 0.000} C_DIS
LIN {X 92.416,Y 274.880,Z 137.642,A -108.583,B 90.000,C 0.000} C_DIS
WAIT SEC 1
RET=EKI_SetBool("oxy","torchState",TRUE)
RET = EKI_Send("oxy","torchState")
LIN {X 92.496,Y 274.854,Z 137.993,A -108.599,B 90.000,C 0.000} C_DIS
LIN {X 92.509,Y 274.849,Z 140.493,A -108.602,B 90.000,C 0.000} C_DIS
LIN {X 92.501,Y 274.852,Z 142.993,A -108.601,B 90.000,C 0.000} C_DIS
LIN {X 92.546,Y 274.837,Z 145.492,A -108.610,B 90.000,C 0.000} C_DIS
LIN {X 92.567,Y 274.830,Z 146.330,A -108.614,B 90.000,C 0.000} C_DIS
LIN {X 92.774,Y 274.760,Z 147.150,A -108.657,B 90.000,C 0.000} C_DIS
LIN {X 93.078,Y 274.657,Z 147.727,A -108.721,B 90.000,C 0.000} C_DIS
LIN {X 93.473,Y 274.523,Z 148.053,A -108.803,B 90.000,C 0.000} C_DIS
LIN {X 93.953,Y 274.359,Z 148.120,A -108.904,B 90.000,C 0.000} C_DIS
LIN {X 94.366,Y 274.217,Z 147.995,A -108.990,B 90.000,C 0.000} C_DIS
LIN {X 94.754,Y 274.083,Z 147.733,A -109.071,B 90.000,C 0.000} C_DIS
LIN {X 95.107,Y 273.961,Z 147.346,A -109.145,B 90.000,C 0.000} C_DIS
LIN {X 95.412,Y 273.855,Z 146.842,A -109.208,B 90.000,C 0.000} C_DIS
LIN {X 95.640,Y 273.775,Z 146.281,A -109.256,B 90.000,C 0.000} C_DIS
LIN {X 95.754,Y 273.736,Z 145.496,A -109.280,B 90.000,C 0.000} C_DIS
LIN {X 95.749,Y 273.737,Z 142.996,A -109.279,B 90.000,C 0.000} C_DIS
LIN {X 95.751,Y 273.737,Z 140.496,A -109.279,B 90.000,C 0.000} C_DIS
LIN {X 95.758,Y 273.734,Z 138.751,A -109.281,B 90.000,C 0.000} C_DIS
LIN {X 97.996,Y 272.941,Z 139.421,A -109.750,B 90.000,C 0.000} C_DIS
LIN {X 98.035,Y 272.927,Z 141.920,A -109.758,B 90.000,C 0.000} C_DIS
LIN {X 98.043,Y 272.924,Z 144.420,A -109.760,B 90.000,C 0.000} C_DIS
LIN {X 98.050,Y 272.921,Z 146.920,A -109.761,B 90.000,C 0.000} C_DIS
LIN {X 98.026,Y 272.930,Z 149.420,A -109.756,B 90.000,C 0.000} C_DIS
LIN {X 98.001,Y 272.939,Z 151.920,A -109.751,B 90.000,C 0.000} C_DIS
LIN {X 97.997,Y 272.941,Z 152.341,A -109.750,B 90.000,C 0.000} C_DIS
LIN {X 97.874,Y 272.985,Z 153.166,A -109.725,B 90.000,C 0.000} C_DIS
LIN {X 97.623,Y 273.075,Z 153.743,A -109.672,B 90.000,C 0.000} C_DIS
LIN {X 97.180,Y 273.233,Z 154.505,A -109.579,B 90.000,C 0.000} C_DIS
LIN {X 96.629,Y 273.428,Z 155.122,A -109.463,B 90.000,C 0.000} C_DIS
LIN {X 95.983,Y 273.655,Z 155.584,A -109.328,B 90.000,C 0.000} C_DIS
LIN {X 95.255,Y 273.910,Z 155.878,A -109.176,B 90.000,C 0.000} C_DIS
LIN {X 94.647,Y 274.120,Z 155.981,A -109.049,B 90.000,C 0.000} C_DIS
LIN {X 94.045,Y 274.327,Z 155.962,A -108.923,B 90.000,C 0.000} C_DIS
LIN {X 93.453,Y 274.530,Z 155.822,A -108.799,B 90.000,C 0.000} C_DIS
LIN {X 92.873,Y 274.726,Z 155.563,A -108.678,B 90.000,C 0.000} C_DIS
LIN {X 92.308,Y 274.917,Z 155.187,A -108.560,B 90.000,C 0.000} C_DIS
LIN {X 91.763,Y 275.099,Z 154.696,A -108.447,B 90.000,C 0.000} C_DIS
LIN {X 90.741,Y 275.438,Z 153.373,A -108.234,B 90.000,C 0.000} C_DIS
LIN {X 89.578,Y 275.818,Z 151.193,A -107.992,B 90.000,C 0.000} C_DIS
LIN {X 89.091,Y 275.976,Z 149.932,A -107.891,B 90.000,C 0.000} C_DIS
LIN {X 88.817,Y 276.064,Z 148.872,A -107.834,B 90.000,C 0.000} C_DIS
LIN {X 88.599,Y 276.134,Z 146.383,A -107.789,B 90.000,C 0.000} C_DIS
LIN {X 88.464,Y 276.178,Z 143.887,A -107.761,B 90.000,C 0.000} C_DIS
LIN {X 88.323,Y 276.223,Z 141.392,A -107.732,B 90.000,C 0.000} C_DIS
LIN {X 88.193,Y 276.264,Z 138.895,A -107.705,B 90.000,C 0.000} C_DIS
LIN {X 88.095,Y 276.296,Z 136.398,A -107.684,B 90.000,C 0.000} C_DIS
LIN {X 88.086,Y 276.298,Z 136.194,A -107.683,B 90.000,C 0.000} C_DIS
LIN {X 90.360,Y 275.558,Z 136.924,A -108.155,B 90.000,C 0.000} C_DIS
LIN {X 92.416,Y 274.880,Z 137.642,A -108.583,B 90.000,C 0.000} C_DIS
LIN {X 91.779,Y 272.985,Z 137.642,A -108.583,B 90.000,C 0.000} C_DIS
WAIT SEC 0.1
RET=EKI_SetBool("oxy","torchState",FALSE)
RET = EKI_Send("oxy","torchState")
LIN {X 86.043,Y 255.923,Z 137.642,A -108.583,B 90.000,C 0.000} C_DIS
LIN {X 99.501,Y 250.997,Z 143.819,A -111.625,B 90.000,C 0.000} C_DIS
LIN {X 106.135,Y 267.730,Z 143.819,A -111.625,B 90.000,C 0.000} C_DIS
LIN {X 106.872,Y 269.589,Z 143.819,A -111.625,B 90.000,C 0.000} C_DIS
WAIT SEC 1
RET=EKI_SetBool("oxy","torchState",TRUE)
RET = EKI_Send("oxy","torchState")
LIN {X 107.896,Y 269.181,Z 145.126,A -111.843,B 90.000,C 0.000} C_DIS
LIN {X 108.080,Y 269.107,Z 145.671,A -111.882,B 90.000,C 0.000} C_DIS
LIN {X 107.985,Y 269.145,Z 148.168,A -111.861,B 90.000,C 0.000} C_DIS
LIN {X 107.909,Y 269.176,Z 150.667,A -111.845,B 90.000,C 0.000} C_DIS
LIN {X 107.882,Y 269.187,Z 153.167,A -111.839,B 90.000,C 0.000} C_DIS
LIN {X 107.850,Y 269.200,Z 155.666,A -111.833,B 90.000,C 0.000} C_DIS
LIN {X 107.800,Y 269.220,Z 158.166,A -111.822,B 90.000,C 0.000} C_DIS
LIN {X 107.750,Y 269.240,Z 160.665,A -111.811,B 90.000,C 0.000} C_DIS
LIN {X 107.701,Y 269.259,Z 163.164,A -111.801,B 90.000,C 0.000} C_DIS
LIN {X 107.661,Y 269.275,Z 165.664,A -111.792,B 90.000,C 0.000} C_DIS
LIN {X 107.620,Y 269.291,Z 168.164,A -111.784,B 90.000,C 0.000} C_DIS
LIN {X 107.582,Y 269.307,Z 170.663,A -111.776,B 90.000,C 0.000} C_DIS
LIN {X 107.547,Y 269.321,Z 173.163,A -111.768,B 90.000,C 0.000} C_DIS
LIN {X 107.513,Y 269.334,Z 175.662,A -111.761,B 90.000,C 0.000} C_DIS
LIN {X 107.519,Y 269.332,Z 177.773,A -111.762,B 90.000,C 0.000} C_DIS
LIN {X 109.836,Y 268.394,Z 177.824,A -112.256,B 90.000,C 0.000} C_DIS
LIN {X 111.480,Y 267.717,Z 177.858,A -112.607,B 90.000,C 0.000} C_DIS
LIN {X 111.389,Y 267.754,Z 178.072,A -112.588,B 90.000,C 0.000} C_DIS
LIN {X 111.036,Y 267.901,Z 178.342,A -112.512,B 90.000,C 0.000} C_DIS
LIN {X 108.857,Y 268.793,Z 179.183,A -112.047,B 90.000,C 0.000} C_DIS
LIN {X 108.397,Y 268.980,Z 179.352,A -111.949,B 90.000,C 0.000} C_DIS
LIN {X 109.075,Y 268.705,Z 181.742,A -112.094,B 90.000,C 0.000} C_DIS
LIN {X 109.752,Y 268.429,Z 184.133,A -112.238,B 90.000,C 0.000} C_DIS
LIN {X 110.129,Y 268.275,Z 185.464,A -112.319,B 90.000,C 0.000} C_DIS
LIN {X 107.828,Y 269.208,Z 185.752,A -111.828,B 90.000,C 0.000} C_DIS
LIN {X 107.138,Y 269.484,Z 185.838,A -111.681,B 90.000,C 0.000} C_DIS
LIN {X 106.922,Y 269.569,Z 183.348,A -111.635,B 90.000,C 0.000} C_DIS
LIN {X 106.700,Y 269.657,Z 180.860,A -111.588,B 90.000,C 0.000} C_DIS
LIN {X 106.564,Y 269.711,Z 179.334,A -111.559,B 90.000,C 0.000} C_DIS
LIN {X 106.485,Y 269.742,Z 179.093,A -111.542,B 90.000,C 0.000} C_DIS
LIN {X 106.180,Y 269.862,Z 178.844,A -111.478,B 90.000,C 0.000} C_DIS
LIN {X 104.512,Y 270.513,Z 177.821,A -111.124,B 90.000,C 0.000} C_DIS
LIN {X 104.651,Y 270.459,Z 175.326,A -111.153,B 90.000,C 0.000} C_DIS
LIN {X 104.798,Y 270.402,Z 172.831,A -111.184,B 90.000,C 0.000} C_DIS
LIN {X 104.945,Y 270.345,Z 170.336,A -111.216,B 90.000,C 0.000} C_DIS
LIN {X 105.092,Y 270.288,Z 167.841,A -111.247,B 90.000,C 0.000} C_DIS
LIN {X 105.239,Y 270.230,Z 165.346,A -111.278,B 90.000,C 0.000} C_DIS
LIN {X 105.386,Y 270.173,Z 162.851,A -111.309,B 90.000,C 0.000} C_DIS
LIN {X 105.533,Y 270.116,Z 160.356,A -111.340,B 90.000,C 0.000} C_DIS
LIN {X 105.684,Y 270.057,Z 157.862,A -111.372,B 90.000,C 0.000} C_DIS
LIN {X 105.848,Y 269.993,Z 155.368,A -111.407,B 90.000,C 0.000} C_DIS
LIN {X 106.011,Y 269.928,Z 152.874,A -111.442,B 90.000,C 0.000} C_DIS
LIN {X 106.175,Y 269.864,Z 150.381,A -111.477,B 90.000,C 0.000} C_DIS
LIN {X 106.339,Y 269.800,Z 147.887,A -111.511,B 90.000,C 0.000} C_DIS
LIN {X 106.502,Y 269.735,Z 145.393,A -111.546,B 90.000,C 0.000} C_DIS
LIN {X 106.620,Y 269.689,Z 143.596,A -111.571,B 90.000,C 0.000} C_DIS
LIN {X 106.872,Y 269.589,Z 143.820,A -111.625,B 90.000,C 0.000} C_DIS
LIN {X 106.135,Y 267.730,Z 143.820,A -111.625,B 90.000,C 0.000} C_DIS
WAIT SEC 0.1
RET=EKI_SetBool("oxy","torchState",FALSE)
RET = EKI_Send("oxy","torchState")
LIN {X 99.501,Y 250.997,Z 143.820,A -111.625,B 90.000,C 0.000} C_DIS
LIN {X 102.329,Y 249.858,Z 141.587,A -112.271,B 90.000,C 0.000} C_DIS
LIN {X 109.150,Y 266.515,Z 141.587,A -112.271,B 90.000,C 0.000} C_DIS
LIN {X 109.908,Y 268.366,Z 141.587,A -112.271,B 90.000,C 0.000} C_DIS
WAIT SEC 1
RET=EKI_SetBool("oxy","torchState",TRUE)
RET = EKI_Send("oxy","torchState")
LIN {X 110.181,Y 268.254,Z 141.704,A -112.330,B 90.000,C 0.000} C_DIS
LIN {X 110.994,Y 267.918,Z 141.764,A -112.503,B 90.000,C 0.000} C_DIS
LIN {X 113.293,Y 266.947,Z 141.616,A -112.997,B 90.000,C 0.000} C_DIS
LIN {X 115.587,Y 265.968,Z 141.442,A -113.489,B 90.000,C 0.000} C_DIS
LIN {X 117.861,Y 264.970,Z 141.154,A -113.980,B 90.000,C 0.000} C_DIS
LIN {X 117.895,Y 264.954,Z 141.148,A -113.987,B 90.000,C 0.000} C_DIS
LIN {X 118.456,Y 264.704,Z 140.899,A -114.109,B 90.000,C 0.000} C_DIS
LIN {X 118.868,Y 264.519,Z 140.528,A -114.198,B 90.000,C 0.000} C_DIS
LIN {X 119.249,Y 264.348,Z 139.938,A -114.280,B 90.000,C 0.000} C_DIS
LIN {X 119.490,Y 264.239,Z 139.252,A -114.333,B 90.000,C 0.000} C_DIS
LIN {X 119.580,Y 264.198,Z 138.524,A -114.352,B 90.000,C 0.000} C_DIS
LIN {X 119.505,Y 264.232,Z 137.814,A -114.336,B 90.000,C 0.000} C_DIS
LIN {X 119.262,Y 264.342,Z 137.163,A -114.283,B 90.000,C 0.000} C_DIS
LIN {X 118.860,Y 264.523,Z 136.634,A -114.196,B 90.000,C 0.000} C_DIS
LIN {X 118.573,Y 264.652,Z 136.352,A -114.134,B 90.000,C 0.000} C_DIS
LIN {X 116.288,Y 265.657,Z 136.482,A -113.641,B 90.000,C 0.000} C_DIS
LIN {X 114.000,Y 266.653,Z 136.642,A -113.148,B 90.000,C 0.000} C_DIS
LIN {X 113.403,Y 266.908,Z 136.702,A -113.019,B 90.000,C 0.000} C_DIS
LIN {X 113.134,Y 267.022,Z 137.917,A -112.962,B 90.000,C 0.000} C_DIS
LIN {X 112.819,Y 267.155,Z 138.754,A -112.894,B 90.000,C 0.000} C_DIS
LIN {X 112.387,Y 267.337,Z 139.510,A -112.802,B 90.000,C 0.000} C_DIS
LIN {X 111.865,Y 267.556,Z 140.128,A -112.690,B 90.000,C 0.000} C_DIS
LIN {X 109.919,Y 268.361,Z 141.409,A -112.274,B 90.000,C 0.000} C_DIS
LIN {X 109.908,Y 268.366,Z 141.587,A -112.271,B 90.000,C 0.000} C_DIS
LIN {X 109.150,Y 266.515,Z 141.587,A -112.271,B 90.000,C 0.000} C_DIS
WAIT SEC 0.1
RET=EKI_SetBool("oxy","torchState",FALSE)
RET = EKI_Send("oxy","torchState")
LIN {X 102.329,Y 249.858,Z 141.587,A -112.271,B 90.000,C 0.000} C_DIS
LIN {X 106.590,Y 248.070,Z 145.294,A -113.252,B 90.000,C 0.000} C_DIS
LIN {X 113.696,Y 264.608,Z 145.294,A -113.252,B 90.000,C 0.000} C_DIS
LIN {X 114.486,Y 266.445,Z 145.294,A -113.252,B 90.000,C 0.000} C_DIS
WAIT SEC 1
RET=EKI_SetBool("oxy","torchState",TRUE)
RET = EKI_Send("oxy","torchState")
LIN {X 114.897,Y 266.268,Z 145.294,A -113.341,B 90.000,C 0.000} C_DIS
LIN {X 116.817,Y 265.431,Z 144.998,A -113.754,B 90.000,C 0.000} C_DIS
LIN {X 117.254,Y 265.238,Z 147.452,A -113.849,B 90.000,C 0.000} C_DIS
LIN {X 117.677,Y 265.050,Z 149.909,A -113.940,B 90.000,C 0.000} C_DIS
LIN {X 118.101,Y 264.861,Z 152.366,A -114.032,B 90.000,C 0.000} C_DIS
LIN {X 118.524,Y 264.673,Z 154.822,A -114.123,B 90.000,C 0.000} C_DIS
LIN {X 118.947,Y 264.483,Z 157.279,A -114.215,B 90.000,C 0.000} C_DIS
LIN {X 119.369,Y 264.292,Z 159.735,A -114.307,B 90.000,C 0.000} C_DIS
LIN {X 119.792,Y 264.101,Z 162.192,A -114.398,B 90.000,C 0.000} C_DIS
LIN {X 120.214,Y 263.910,Z 164.648,A -114.490,B 90.000,C 0.000} C_DIS
LIN {X 120.632,Y 263.718,Z 167.106,A -114.581,B 90.000,C 0.000} C_DIS
LIN {X 121.050,Y 263.527,Z 169.563,A -114.672,B 90.000,C 0.000} C_DIS
LIN {X 121.468,Y 263.335,Z 172.020,A -114.762,B 90.000,C 0.000} C_DIS
LIN {X 121.868,Y 263.150,Z 174.481,A -114.849,B 90.000,C 0.000} C_DIS
LIN {X 122.245,Y 262.975,Z 176.946,A -114.932,B 90.000,C 0.000} C_DIS
LIN {X 122.325,Y 262.938,Z 177.467,A -114.949,B 90.000,C 0.000} C_DIS
LIN {X 122.158,Y 263.016,Z 177.555,A -114.912,B 90.000,C 0.000} C_DIS
LIN {X 121.002,Y 263.550,Z 177.741,A -114.661,B 90.000,C 0.000} C_DIS
LIN {X 121.199,Y 263.459,Z 180.231,A -114.704,B 90.000,C 0.000} C_DIS
LIN {X 121.215,Y 263.452,Z 180.427,A -114.707,B 90.000,C 0.000} C_DIS
LIN {X 121.387,Y 263.373,Z 181.335,A -114.745,B 90.000,C 0.000} C_DIS
LIN {X 122.082,Y 263.051,Z 183.007,A -114.896,B 90.000,C 0.000} C_DIS
LIN {X 122.161,Y 263.015,Z 183.708,A -114.913,B 90.000,C 0.000} C_DIS
LIN {X 122.055,Y 263.064,Z 185.493,A -114.890,B 90.000,C 0.000} C_DIS
LIN {X 120.129,Y 263.949,Z 185.822,A -114.471,B 90.000,C 0.000} C_DIS
LIN {X 120.045,Y 263.987,Z 186.013,A -114.453,B 90.000,C 0.000} C_DIS
LIN {X 120.065,Y 263.978,Z 186.396,A -114.458,B 90.000,C 0.000} C_DIS
LIN {X 120.211,Y 263.912,Z 187.361,A -114.489,B 90.000,C 0.000} C_DIS
LIN {X 121.079,Y 263.515,Z 189.672,A -114.678,B 90.000,C 0.000} C_DIS
LIN {X 121.242,Y 263.440,Z 190.383,A -114.713,B 90.000,C 0.000} C_DIS
LIN {X 121.263,Y 263.430,Z 190.549,A -114.718,B 90.000,C 0.000} C_DIS
LIN {X 121.351,Y 263.390,Z 190.596,A -114.737,B 90.000,C 0.000} C_DIS
LIN {X 122.685,Y 262.770,Z 189.896,A -115.027,B 90.000,C 0.000} C_DIS
LIN {X 123.211,Y 262.524,Z 189.797,A -115.142,B 90.000,C 0.000} C_DIS
LIN {X 123.403,Y 262.434,Z 189.840,A -115.184,B 90.000,C 0.000} C_DIS
LIN {X 123.450,Y 262.412,Z 190.004,A -115.194,B 90.000,C 0.000} C_DIS
LIN {X 123.349,Y 262.460,Z 190.710,A -115.172,B 90.000,C 0.000} C_DIS
LIN {X 122.616,Y 262.802,Z 193.075,A -115.012,B 90.000,C 0.000} C_DIS
LIN {X 121.834,Y 263.165,Z 195.422,A -114.842,B 90.000,C 0.000} C_DIS
LIN {X 121.029,Y 263.537,Z 197.759,A -114.667,B 90.000,C 0.000} C_DIS
LIN {X 120.166,Y 263.932,Z 200.072,A -114.479,B 90.000,C 0.000} C_DIS
LIN {X 119.277,Y 264.334,Z 202.373,A -114.287,B 90.000,C 0.000} C_DIS
LIN {X 118.369,Y 264.743,Z 204.667,A -114.090,B 90.000,C 0.000} C_DIS
LIN {X 118.198,Y 264.819,Z 205.055,A -114.053,B 90.000,C 0.000} C_DIS
LIN {X 118.007,Y 264.904,Z 204.775,A -114.012,B 90.000,C 0.000} C_DIS
LIN {X 117.425,Y 265.163,Z 203.573,A -113.886,B 90.000,C 0.000} C_DIS
LIN {X 116.653,Y 265.503,Z 201.219,A -113.719,B 90.000,C 0.000} C_DIS
LIN {X 115.973,Y 265.800,Z 198.832,A -113.572,B 90.000,C 0.000} C_DIS
LIN {X 115.324,Y 266.083,Z 196.435,A -113.433,B 90.000,C 0.000} C_DIS
LIN {X 114.783,Y 266.317,Z 194.005,A -113.316,B 90.000,C 0.000} C_DIS
LIN {X 114.445,Y 266.463,Z 192.054,A -113.243,B 90.000,C 0.000} C_DIS
LIN {X 114.491,Y 266.443,Z 191.419,A -113.253,B 90.000,C 0.000} C_DIS
LIN {X 115.196,Y 266.139,Z 190.543,A -113.405,B 90.000,C 0.000} C_DIS
LIN {X 116.192,Y 265.706,Z 188.291,A -113.620,B 90.000,C 0.000} C_DIS
LIN {X 116.537,Y 265.554,Z 187.531,A -113.694,B 90.000,C 0.000} C_DIS
LIN {X 117.598,Y 265.086,Z 186.581,A -113.923,B 90.000,C 0.000} C_DIS
LIN {X 117.856,Y 264.972,Z 186.236,A -113.979,B 90.000,C 0.000} C_DIS
LIN {X 117.903,Y 264.951,Z 186.120,A -113.989,B 90.000,C 0.000} C_DIS
LIN {X 117.856,Y 264.972,Z 186.027,A -113.979,B 90.000,C 0.000} C_DIS
LIN {X 116.689,Y 265.488,Z 185.394,A -113.727,B 90.000,C 0.000} C_DIS
LIN {X 116.435,Y 265.599,Z 185.142,A -113.672,B 90.000,C 0.000} C_DIS
LIN {X 116.407,Y 265.612,Z 184.869,A -113.666,B 90.000,C 0.000} C_DIS
LIN {X 116.698,Y 265.484,Z 184.257,A -113.729,B 90.000,C 0.000} C_DIS
LIN {X 116.727,Y 265.471,Z 183.933,A -113.735,B 90.000,C 0.000} C_DIS
LIN {X 116.647,Y 265.506,Z 183.200,A -113.718,B 90.000,C 0.000} C_DIS
LIN {X 116.025,Y 265.778,Z 180.794,A -113.584,B 90.000,C 0.000} C_DIS
LIN {X 115.581,Y 265.972,Z 178.647,A -113.488,B 90.000,C 0.000} C_DIS
LIN {X 115.549,Y 265.986,Z 177.760,A -113.481,B 90.000,C 0.000} C_DIS
LIN {X 115.585,Y 265.970,Z 177.554,A -113.489,B 90.000,C 0.000} C_DIS
LIN {X 117.873,Y 264.964,Z 177.554,A -113.983,B 90.000,C 0.000} C_DIS
LIN {X 117.930,Y 264.939,Z 177.554,A -113.995,B 90.000,C 0.000} C_DIS
LIN {X 117.671,Y 265.054,Z 175.070,A -113.939,B 90.000,C 0.000} C_DIS
LIN {X 117.408,Y 265.170,Z 172.587,A -113.882,B 90.000,C 0.000} C_DIS
LIN {X 117.145,Y 265.286,Z 170.104,A -113.825,B 90.000,C 0.000} C_DIS
LIN {X 116.882,Y 265.402,Z 167.620,A -113.769,B 90.000,C 0.000} C_DIS
LIN {X 116.619,Y 265.517,Z 165.137,A -113.712,B 90.000,C 0.000} C_DIS
LIN {X 116.356,Y 265.633,Z 162.654,A -113.655,B 90.000,C 0.000} C_DIS
LIN {X 116.091,Y 265.749,Z 160.170,A -113.598,B 90.000,C 0.000} C_DIS
LIN {X 115.825,Y 265.865,Z 157.687,A -113.540,B 90.000,C 0.000} C_DIS
LIN {X 115.558,Y 265.981,Z 155.204,A -113.483,B 90.000,C 0.000} C_DIS
LIN {X 115.291,Y 266.097,Z 152.722,A -113.425,B 90.000,C 0.000} C_DIS
LIN {X 115.024,Y 266.212,Z 150.239,A -113.368,B 90.000,C 0.000} C_DIS
LIN {X 114.757,Y 266.328,Z 147.756,A -113.311,B 90.000,C 0.000} C_DIS
LIN {X 114.486,Y 266.445,Z 145.294,A -113.252,B 90.000,C 0.000} C_DIS
LIN {X 113.696,Y 264.608,Z 145.294,A -113.252,B 90.000,C 0.000} C_DIS
WAIT SEC 0.1
RET=EKI_SetBool("oxy","torchState",FALSE)
RET = EKI_Send("oxy","torchState")
LIN {X 106.590,Y 248.070,Z 145.294,A -113.252,B 90.000,C 0.000} C_DIS
LIN {X 86.211,Y 255.867,Z 157.799,A -108.620,B 90.000,C 0.000} C_DIS
LIN {X 91.958,Y 272.924,Z 157.799,A -108.620,B 90.000,C 0.000} C_DIS
LIN {X 92.596,Y 274.820,Z 157.799,A -108.620,B 90.000,C 0.000} C_DIS
WAIT SEC 1
RET=EKI_SetBool("oxy","torchState",TRUE)
RET = EKI_Send("oxy","torchState")
LIN {X 94.592,Y 274.139,Z 159.142,A -109.037,B 90.000,C 0.000} C_DIS
LIN {X 94.739,Y 274.088,Z 159.243,A -109.068,B 90.000,C 0.000} C_DIS
LIN {X 94.805,Y 274.066,Z 161.742,A -109.082,B 90.000,C 0.000} C_DIS
LIN {X 94.854,Y 274.049,Z 164.241,A -109.092,B 90.000,C 0.000} C_DIS
LIN {X 94.904,Y 274.032,Z 166.741,A -109.102,B 90.000,C 0.000} C_DIS
LIN {X 94.953,Y 274.014,Z 169.240,A -109.113,B 90.000,C 0.000} C_DIS
LIN {X 95.003,Y 273.997,Z 171.739,A -109.123,B 90.000,C 0.000} C_DIS
LIN {X 95.052,Y 273.980,Z 174.239,A -109.133,B 90.000,C 0.000} C_DIS
LIN {X 95.102,Y 273.963,Z 176.738,A -109.144,B 90.000,C 0.000} C_DIS
LIN {X 95.151,Y 273.946,Z 179.237,A -109.154,B 90.000,C 0.000} C_DIS
LIN {X 95.201,Y 273.928,Z 181.737,A -109.164,B 90.000,C 0.000} C_DIS
LIN {X 95.248,Y 273.912,Z 184.236,A -109.174,B 90.000,C 0.000} C_DIS
LIN {X 95.296,Y 273.895,Z 186.735,A -109.184,B 90.000,C 0.000} C_DIS
LIN {X 95.343,Y 273.879,Z 189.235,A -109.194,B 90.000,C 0.000} C_DIS
LIN {X 95.390,Y 273.863,Z 191.734,A -109.204,B 90.000,C 0.000} C_DIS
LIN {X 95.437,Y 273.846,Z 194.234,A -109.214,B 90.000,C 0.000} C_DIS
LIN {X 95.485,Y 273.830,Z 196.733,A -109.224,B 90.000,C 0.000} C_DIS
LIN {X 95.532,Y 273.813,Z 199.233,A -109.234,B 90.000,C 0.000} C_DIS
LIN {X 95.579,Y 273.797,Z 201.732,A -109.243,B 90.000,C 0.000} C_DIS
LIN {X 95.587,Y 273.794,Z 202.147,A -109.245,B 90.000,C 0.000} C_DIS
LIN {X 95.622,Y 273.782,Z 204.295,A -109.252,B 90.000,C 0.000} C_DIS
LIN {X 93.512,Y 274.510,Z 204.295,A -108.811,B 90.000,C 0.000} C_DIS
LIN {X 93.446,Y 274.532,Z 201.796,A -108.798,B 90.000,C 0.000} C_DIS
LIN {X 93.365,Y 274.560,Z 199.298,A -108.781,B 90.000,C 0.000} C_DIS
LIN {X 93.283,Y 274.588,Z 196.799,A -108.764,B 90.000,C 0.000} C_DIS
LIN {X 93.201,Y 274.615,Z 194.301,A -108.747,B 90.000,C 0.000} C_DIS
LIN {X 93.119,Y 274.643,Z 191.802,A -108.729,B 90.000,C 0.000} C_DIS
LIN {X 93.036,Y 274.671,Z 189.304,A -108.712,B 90.000,C 0.000} C_DIS
LIN {X 92.953,Y 274.699,Z 186.805,A -108.695,B 90.000,C 0.000} C_DIS
LIN {X 92.871,Y 274.727,Z 184.307,A -108.678,B 90.000,C 0.000} C_DIS
LIN {X 92.788,Y 274.755,Z 181.809,A -108.661,B 90.000,C 0.000} C_DIS
LIN {X 92.706,Y 274.782,Z 179.310,A -108.643,B 90.000,C 0.000} C_DIS
LIN {X 92.623,Y 274.810,Z 176.812,A -108.626,B 90.000,C 0.000} C_DIS
LIN {X 92.540,Y 274.838,Z 174.313,A -108.609,B 90.000,C 0.000} C_DIS
LIN {X 92.458,Y 274.866,Z 171.815,A -108.592,B 90.000,C 0.000} C_DIS
LIN {X 92.375,Y 274.894,Z 169.317,A -108.574,B 90.000,C 0.000} C_DIS
LIN {X 92.293,Y 274.921,Z 166.818,A -108.557,B 90.000,C 0.000} C_DIS
LIN {X 92.210,Y 274.949,Z 164.320,A -108.540,B 90.000,C 0.000} C_DIS
LIN {X 92.127,Y 274.977,Z 161.821,A -108.523,B 90.000,C 0.000} C_DIS
LIN {X 92.045,Y 275.005,Z 159.323,A -108.506,B 90.000,C 0.000} C_DIS
LIN {X 91.985,Y 275.025,Z 157.584,A -108.493,B 90.000,C 0.000} C_DIS
LIN {X 92.116,Y 274.981,Z 157.584,A -108.520,B 90.000,C 0.000} C_DIS
LIN {X 92.596,Y 274.820,Z 157.800,A -108.620,B 90.000,C 0.000} C_DIS
LIN {X 91.958,Y 272.924,Z 157.800,A -108.620,B 90.000,C 0.000} C_DIS
WAIT SEC 0.1
RET=EKI_SetBool("oxy","torchState",FALSE)
RET = EKI_Send("oxy","torchState")
LIN {X 86.210,Y 255.867,Z 157.800,A -108.620,B 90.000,C 0.000} C_DIS
LIN {X 99.477,Y 251.007,Z 187.401,A -111.619,B 90.000,C 0.000} C_DIS
LIN {X 106.109,Y 267.740,Z 187.401,A -111.619,B 90.000,C 0.000} C_DIS
LIN {X 106.846,Y 269.600,Z 187.401,A -111.619,B 90.000,C 0.000} C_DIS
WAIT SEC 1
RET=EKI_SetBool("oxy","torchState",TRUE)
RET = EKI_Send("oxy","torchState")
LIN {X 107.669,Y 269.272,Z 189.738,A -111.794,B 90.000,C 0.000} C_DIS
LIN {X 108.653,Y 268.873,Z 192.002,A -112.004,B 90.000,C 0.000} C_DIS
LIN {X 109.691,Y 268.450,Z 194.236,A -112.225,B 90.000,C 0.000} C_DIS
LIN {X 110.729,Y 268.027,Z 196.471,A -112.447,B 90.000,C 0.000} C_DIS
LIN {X 111.763,Y 267.595,Z 198.705,A -112.668,B 90.000,C 0.000} C_DIS
LIN {X 112.796,Y 267.161,Z 200.940,A -112.890,B 90.000,C 0.000} C_DIS
LIN {X 113.839,Y 266.722,Z 203.169,A -113.113,B 90.000,C 0.000} C_DIS
LIN {X 114.931,Y 266.253,Z 205.369,A -113.348,B 90.000,C 0.000} C_DIS
LIN {X 115.706,Y 265.918,Z 206.801,A -113.515,B 90.000,C 0.000} C_DIS
LIN {X 115.963,Y 265.805,Z 207.071,A -113.570,B 90.000,C 0.000} C_DIS
LIN {X 116.209,Y 265.698,Z 207.140,A -113.623,B 90.000,C 0.000} C_DIS
LIN {X 116.624,Y 265.516,Z 207.047,A -113.713,B 90.000,C 0.000} C_DIS
LIN {X 116.800,Y 265.439,Z 206.942,A -113.751,B 90.000,C 0.000} C_DIS
LIN {X 116.802,Y 265.438,Z 206.777,A -113.751,B 90.000,C 0.000} C_DIS
LIN {X 115.976,Y 265.799,Z 204.445,A -113.573,B 90.000,C 0.000} C_DIS
LIN {X 115.073,Y 266.192,Z 202.147,A -113.379,B 90.000,C 0.000} C_DIS
LIN {X 114.165,Y 266.580,Z 199.851,A -113.183,B 90.000,C 0.000} C_DIS
LIN {X 113.257,Y 266.968,Z 197.554,A -112.988,B 90.000,C 0.000} C_DIS
LIN {X 112.378,Y 267.340,Z 195.244,A -112.800,B 90.000,C 0.000} C_DIS
LIN {X 111.599,Y 267.667,Z 193.134,A -112.633,B 90.000,C 0.000} C_DIS
LIN {X 111.397,Y 267.751,Z 192.326,A -112.590,B 90.000,C 0.000} C_DIS
LIN {X 111.309,Y 267.788,Z 191.589,A -112.571,B 90.000,C 0.000} C_DIS
LIN {X 111.334,Y 267.777,Z 190.866,A -112.576,B 90.000,C 0.000} C_DIS
LIN {X 111.469,Y 267.721,Z 190.101,A -112.605,B 90.000,C 0.000} C_DIS
LIN {X 111.818,Y 267.576,Z 189.086,A -112.680,B 90.000,C 0.000} C_DIS
LIN {X 112.362,Y 267.348,Z 188.254,A -112.796,B 90.000,C 0.000} C_DIS
LIN {X 112.729,Y 267.193,Z 187.824,A -112.875,B 90.000,C 0.000} C_DIS
LIN {X 110.422,Y 268.154,Z 187.754,A -112.381,B 90.000,C 0.000} C_DIS
LIN {X 108.129,Y 269.088,Z 187.700,A -111.892,B 90.000,C 0.000} C_DIS
LIN {X 107.096,Y 269.500,Z 187.489,A -111.672,B 90.000,C 0.000} C_DIS
LIN {X 106.846,Y 269.600,Z 187.401,A -111.619,B 90.000,C 0.000} C_DIS
LIN {X 106.109,Y 267.740,Z 187.401,A -111.619,B 90.000,C 0.000} C_DIS
WAIT SEC 0.1
RET=EKI_SetBool("oxy","torchState",FALSE)
RET = EKI_Send("oxy","torchState")
LIN {X 99.477,Y 251.007,Z 187.401,A -111.619,B 90.000,C 0.000} C_DIS
LIN {X 89.076,Y 254.883,Z 209.069,A -109.263,B 90.000,C 0.000} C_DIS
LIN {X 95.015,Y 271.875,Z 209.069,A -109.263,B 90.000,C 0.000} C_DIS
LIN {X 95.675,Y 273.763,Z 209.069,A -109.263,B 90.000,C 0.000} C_DIS
WAIT SEC 1
RET=EKI_SetBool("oxy","torchState",TRUE)
RET = EKI_Send("oxy","torchState")
LIN {X 95.005,Y 273.996,Z 208.799,A -109.123,B 90.000,C 0.000} C_DIS
LIN {X 94.318,Y 274.234,Z 208.627,A -108.980,B 90.000,C 0.000} C_DIS
LIN {X 93.781,Y 274.418,Z 208.570,A -108.868,B 90.000,C 0.000} C_DIS
LIN {X 92.344,Y 274.905,Z 208.752,A -108.568,B 90.000,C 0.000} C_DIS
LIN {X 92.487,Y 274.856,Z 209.299,A -108.598,B 90.000,C 0.000} C_DIS
LIN {X 92.827,Y 274.742,Z 210.127,A -108.669,B 90.000,C 0.000} C_DIS
LIN {X 94.029,Y 274.332,Z 212.281,A -108.919,B 90.000,C 0.000} C_DIS
LIN {X 94.446,Y 274.190,Z 213.028,A -109.007,B 90.000,C 0.000} C_DIS
LIN {X 94.896,Y 274.034,Z 213.629,A -109.101,B 90.000,C 0.000} C_DIS
LIN {X 95.319,Y 273.887,Z 214.027,A -109.189,B 90.000,C 0.000} C_DIS
LIN {X 97.558,Y 273.096,Z 214.808,A -109.658,B 90.000,C 0.000} C_DIS
LIN {X 97.905,Y 272.974,Z 214.929,A -109.731,B 90.000,C 0.000} C_DIS
LIN {X 98.561,Y 272.738,Z 214.991,A -109.869,B 90.000,C 0.000} C_DIS
LIN {X 98.879,Y 272.622,Z 214.969,A -109.935,B 90.000,C 0.000} C_DIS
LIN {X 99.037,Y 272.565,Z 214.881,A -109.969,B 90.000,C 0.000} C_DIS
LIN {X 99.278,Y 272.477,Z 214.455,A -110.019,B 90.000,C 0.000} C_DIS
LIN {X 99.324,Y 272.461,Z 213.893,A -110.029,B 90.000,C 0.000} C_DIS
LIN {X 99.174,Y 272.515,Z 213.185,A -109.998,B 90.000,C 0.000} C_DIS
LIN {X 98.828,Y 272.641,Z 212.323,A -109.925,B 90.000,C 0.000} C_DIS
LIN {X 97.998,Y 272.940,Z 210.973,A -109.750,B 90.000,C 0.000} C_DIS
LIN {X 96.924,Y 273.323,Z 209.869,A -109.525,B 90.000,C 0.000} C_DIS
LIN {X 95.675,Y 273.763,Z 209.069,A -109.263,B 90.000,C 0.000} C_DIS
LIN {X 95.015,Y 271.875,Z 209.069,A -109.263,B 90.000,C 0.000} C_DIS
WAIT SEC 0.1
RET=EKI_SetBool("oxy","torchState",FALSE)
RET = EKI_Send("oxy","torchState")
LIN {X 89.076,Y 254.883,Z 209.069,A -109.263,B 90.000,C 0.000} C_DIS
LIN {X 85.319,Y 256.165,Z 211.140,A -108.421,B 90.000,C 0.000} C_DIS
LIN {X 91.007,Y 273.243,Z 211.140,A -108.421,B 90.000,C 0.000} C_DIS
LIN {X 91.639,Y 275.141,Z 211.140,A -108.421,B 90.000,C 0.000} C_DIS
WAIT SEC 1
RET=EKI_SetBool("oxy","torchState",TRUE)
RET = EKI_Send("oxy","torchState")
LIN {X 90.315,Y 275.577,Z 209.064,A -108.146,B 90.000,C 0.000} C_DIS
LIN {X 90.032,Y 275.670,Z 208.621,A -108.087,B 90.000,C 0.000} C_DIS
LIN {X 89.121,Y 275.966,Z 207.584,A -107.897,B 90.000,C 0.000} C_DIS
LIN {X 88.682,Y 276.108,Z 207.243,A -107.806,B 90.000,C 0.000} C_DIS
LIN {X 88.259,Y 276.243,Z 207.025,A -107.719,B 90.000,C 0.000} C_DIS
LIN {X 87.836,Y 276.378,Z 206.919,A -107.631,B 90.000,C 0.000} C_DIS
LIN {X 87.437,Y 276.504,Z 206.929,A -107.548,B 90.000,C 0.000} C_DIS
LIN {X 87.073,Y 276.619,Z 207.053,A -107.473,B 90.000,C 0.000} C_DIS
LIN {X 86.751,Y 276.721,Z 207.289,A -107.406,B 90.000,C 0.000} C_DIS
LIN {X 86.436,Y 276.819,Z 207.706,A -107.341,B 90.000,C 0.000} C_DIS
LIN {X 86.260,Y 276.874,Z 208.195,A -107.304,B 90.000,C 0.000} C_DIS
LIN {X 86.227,Y 276.884,Z 208.738,A -107.298,B 90.000,C 0.000} C_DIS
LIN {X 86.472,Y 276.808,Z 209.864,A -107.348,B 90.000,C 0.000} C_DIS
LIN {X 86.393,Y 276.833,Z 210.292,A -107.332,B 90.000,C 0.000} C_DIS
LIN {X 86.179,Y 276.899,Z 210.693,A -107.288,B 90.000,C 0.000} C_DIS
LIN {X 85.785,Y 277.021,Z 211.082,A -107.206,B 90.000,C 0.000} C_DIS
LIN {X 83.683,Y 277.661,Z 212.274,A -106.772,B 90.000,C 0.000} C_DIS
LIN {X 81.550,Y 278.295,Z 213.413,A -106.332,B 90.000,C 0.000} C_DIS
LIN {X 79.403,Y 278.912,Z 214.536,A -105.891,B 90.000,C 0.000} C_DIS
LIN {X 77.216,Y 279.530,Z 215.576,A -105.442,B 90.000,C 0.000} C_DIS
LIN {X 74.941,Y 280.149,Z 216.408,A -104.976,B 90.000,C 0.000} C_DIS
LIN {X 74.030,Y 280.392,Z 216.770,A -104.790,B 90.000,C 0.000} C_DIS
LIN {X 73.763,Y 280.462,Z 217.015,A -104.735,B 90.000,C 0.000} C_DIS
LIN {X 73.686,Y 280.482,Z 217.293,A -104.720,B 90.000,C 0.000} C_DIS
LIN {X 73.834,Y 280.443,Z 217.625,A -104.750,B 90.000,C 0.000} C_DIS
LIN {X 74.292,Y 280.322,Z 217.866,A -104.843,B 90.000,C 0.000} C_DIS
LIN {X 75.079,Y 280.113,Z 218.023,A -105.004,B 90.000,C 0.000} C_DIS
LIN {X 77.490,Y 279.452,Z 218.053,A -105.498,B 90.000,C 0.000} C_DIS
LIN {X 79.888,Y 278.775,Z 217.851,A -105.991,B 90.000,C 0.000} C_DIS
LIN {X 82.264,Y 278.085,Z 217.495,A -106.479,B 90.000,C 0.000} C_DIS
LIN {X 84.613,Y 277.379,Z 217.014,A -106.964,B 90.000,C 0.000} C_DIS
LIN {X 86.932,Y 276.658,Z 216.420,A -107.444,B 90.000,C 0.000} C_DIS
LIN {X 89.229,Y 275.929,Z 215.754,A -107.920,B 90.000,C 0.000} C_DIS
LIN {X 91.425,Y 275.212,Z 215.006,A -108.377,B 90.000,C 0.000} C_DIS
LIN {X 92.292,Y 274.922,Z 214.586,A -108.557,B 90.000,C 0.000} C_DIS
LIN {X 93.130,Y 274.639,Z 213.963,A -108.732,B 90.000,C 0.000} C_DIS
LIN {X 91.985,Y 275.024,Z 211.775,A -108.493,B 90.000,C 0.000} C_DIS
LIN {X 91.639,Y 275.141,Z 211.140,A -108.421,B 90.000,C 0.000} C_DIS
LIN {X 91.007,Y 273.243,Z 211.140,A -108.421,B 90.000,C 0.000} C_DIS
WAIT SEC 0.1
RET=EKI_SetBool("oxy","torchState",FALSE)
RET = EKI_Send("oxy","torchState")
LIN {X 85.319,Y 256.165,Z 211.140,A -108.421,B 90.000,C 0.000} C_DIS
LIN {X 75.089,Y 259.348,Z 211.974,A -106.147,B 90.000,C 0.000} C_DIS
LIN {X 80.095,Y 276.638,Z 211.974,A -106.147,B 90.000,C 0.000} C_DIS
LIN {X 80.651,Y 278.559,Z 211.974,A -106.147,B 90.000,C 0.000} C_DIS
WAIT SEC 1
RET=EKI_SetBool("oxy","torchState",TRUE)
RET = EKI_Send("oxy","torchState")
LIN {X 80.595,Y 278.576,Z 211.749,A -106.136,B 90.000,C 0.000} C_DIS
LIN {X 80.282,Y 278.666,Z 211.476,A -106.071,B 90.000,C 0.000} C_DIS
LIN {X 79.765,Y 278.814,Z 211.120,A -105.965,B 90.000,C 0.000} C_DIS
LIN {X 79.311,Y 278.944,Z 210.914,A -105.872,B 90.000,C 0.000} C_DIS
LIN {X 78.672,Y 279.125,Z 210.857,A -105.741,B 90.000,C 0.000} C_DIS
LIN {X 77.887,Y 279.345,Z 211.058,A -105.579,B 90.000,C 0.000} C_DIS
LIN {X 77.149,Y 279.550,Z 211.628,A -105.428,B 90.000,C 0.000} C_DIS
LIN {X 76.616,Y 279.696,Z 212.277,A -105.319,B 90.000,C 0.000} C_DIS
LIN {X 76.139,Y 279.826,Z 213.034,A -105.221,B 90.000,C 0.000} C_DIS
LIN {X 75.797,Y 279.919,Z 213.758,A -105.151,B 90.000,C 0.000} C_DIS
LIN {X 75.665,Y 279.955,Z 214.310,A -105.124,B 90.000,C 0.000} C_DIS
LIN {X 75.802,Y 279.918,Z 214.651,A -105.152,B 90.000,C 0.000} C_DIS
LIN {X 76.174,Y 279.817,Z 214.793,A -105.229,B 90.000,C 0.000} C_DIS
LIN {X 76.728,Y 279.666,Z 214.731,A -105.342,B 90.000,C 0.000} C_DIS
LIN {X 77.406,Y 279.479,Z 214.459,A -105.481,B 90.000,C 0.000} C_DIS
LIN {X 79.464,Y 278.900,Z 213.163,A -105.903,B 90.000,C 0.000} C_DIS
LIN {X 80.542,Y 278.591,Z 212.332,A -106.125,B 90.000,C 0.000} C_DIS
LIN {X 80.651,Y 278.559,Z 211.974,A -106.147,B 90.000,C 0.000} C_DIS
LIN {X 80.095,Y 276.638,Z 211.974,A -106.147,B 90.000,C 0.000} C_DIS
WAIT SEC 0.1
RET=EKI_SetBool("oxy","torchState",FALSE)
RET = EKI_Send("oxy","torchState")
LIN {X 75.089,Y 259.348,Z 211.974,A -106.147,B 90.000,C 0.000} C_DIS
LIN {X 69.295,Y 260.956,Z 195.811,A -104.871,B 90.000,C 0.000} C_DIS
LIN {X 73.914,Y 278.354,Z 195.811,A -104.871,B 90.000,C 0.000} C_DIS
LIN {X 74.428,Y 280.287,Z 195.811,A -104.871,B 90.000,C 0.000} C_DIS
WAIT SEC 1
RET=EKI_SetBool("oxy","torchState",TRUE)
RET = EKI_Send("oxy","torchState")
LIN {X 76.675,Y 279.679,Z 194.901,A -105.331,B 90.000,C 0.000} C_DIS
LIN {X 78.848,Y 279.074,Z 193.823,A -105.777,B 90.000,C 0.000} C_DIS
LIN {X 80.923,Y 278.479,Z 192.561,A -106.203,B 90.000,C 0.000} C_DIS
LIN {X 82.064,Y 278.146,Z 191.791,A -106.438,B 90.000,C 0.000} C_DIS
LIN {X 82.595,Y 277.989,Z 191.334,A -106.548,B 90.000,C 0.000} C_DIS
LIN {X 82.780,Y 277.934,Z 191.049,A -106.586,B 90.000,C 0.000} C_DIS
LIN {X 82.669,Y 277.967,Z 190.999,A -106.563,B 90.000,C 0.000} C_DIS
LIN {X 82.354,Y 278.061,Z 191.070,A -106.498,B 90.000,C 0.000} C_DIS
LIN {X 80.118,Y 278.712,Z 191.978,A -106.038,B 90.000,C 0.000} C_DIS
LIN {X 77.840,Y 279.356,Z 192.781,A -105.570,B 90.000,C 0.000} C_DIS
LIN {X 75.525,Y 279.991,Z 193.479,A -105.096,B 90.000,C 0.000} C_DIS
LIN {X 73.176,Y 280.614,Z 194.064,A -104.616,B 90.000,C 0.000} C_DIS
LIN {X 70.799,Y 281.224,Z 194.542,A -104.131,B 90.000,C 0.000} C_DIS
LIN {X 68.400,Y 281.817,Z 194.918,A -103.642,B 90.000,C 0.000} C_DIS
LIN {X 65.983,Y 282.392,Z 195.196,A -103.152,B 90.000,C 0.000} C_DIS
LIN {X 63.553,Y 282.949,Z 195.381,A -102.659,B 90.000,C 0.000} C_DIS
LIN {X 61.113,Y 283.485,Z 195.475,A -102.165,B 90.000,C 0.000} C_DIS
LIN {X 58.667,Y 284.001,Z 195.480,A -101.672,B 90.000,C 0.000} C_DIS
LIN {X 56.217,Y 284.491,Z 195.383,A -101.178,B 90.000,C 0.000} C_DIS
LIN {X 53.768,Y 284.971,Z 195.246,A -100.685,B 90.000,C 0.000} C_DIS
LIN {X 51.321,Y 285.415,Z 194.984,A -100.194,B 90.000,C 0.000} C_DIS
LIN {X 48.878,Y 285.847,Z 194.679,A -99.703,B 90.000,C 0.000} C_DIS
LIN {X 46.444,Y 286.253,Z 194.276,A -99.216,B 90.000,C 0.000} C_DIS
LIN {X 44.029,Y 286.633,Z 193.756,A -98.733,B 90.000,C 0.000} C_DIS
LIN {X 42.375,Y 286.887,Z 193.364,A -98.402,B 90.000,C 0.000} C_DIS
LIN {X 40.166,Y 287.205,Z 192.588,A -97.961,B 90.000,C 0.000} C_DIS
LIN {X 38.443,Y 287.441,Z 191.658,A -97.618,B 90.000,C 0.000} C_DIS
LIN {X 37.768,Y 287.530,Z 191.138,A -97.483,B 90.000,C 0.000} C_DIS
LIN {X 37.220,Y 287.602,Z 190.584,A -97.374,B 90.000,C 0.000} C_DIS
LIN {X 36.802,Y 287.655,Z 189.996,A -97.291,B 90.000,C 0.000} C_DIS
LIN {X 36.514,Y 287.692,Z 189.375,A -97.233,B 90.000,C 0.000} C_DIS
LIN {X 36.322,Y 287.716,Z 188.470,A -97.195,B 90.000,C 0.000} C_DIS
LIN {X 36.317,Y 287.717,Z 185.970,A -97.194,B 90.000,C 0.000} C_DIS
LIN {X 36.311,Y 287.718,Z 184.901,A -97.193,B 90.000,C 0.000} C_DIS
LIN {X 36.158,Y 287.737,Z 184.227,A -97.162,B 90.000,C 0.000} C_DIS
LIN {X 35.872,Y 287.773,Z 183.571,A -97.106,B 90.000,C 0.000} C_DIS
LIN {X 34.571,Y 287.931,Z 181.442,A -96.847,B 90.000,C 0.000} C_DIS
LIN {X 33.161,Y 288.097,Z 179.385,A -96.566,B 90.000,C 0.000} C_DIS
LIN {X 32.605,Y 288.161,Z 178.650,A -96.455,B 90.000,C 0.000} C_DIS
LIN {X 31.258,Y 288.310,Z 177.301,A -96.188,B 90.000,C 0.000} C_DIS
LIN {X 30.126,Y 288.431,Z 176.495,A -95.963,B 90.000,C 0.000} C_DIS
LIN {X 28.904,Y 288.556,Z 175.889,A -95.720,B 90.000,C 0.000} C_DIS
LIN {X 27.593,Y 288.684,Z 175.484,A -95.460,B 90.000,C 0.000} C_DIS
LIN {X 26.191,Y 288.815,Z 175.279,A -95.182,B 90.000,C 0.000} C_DIS
LIN {X 23.853,Y 289.017,Z 175.341,A -94.718,B 90.000,C 0.000} C_DIS
LIN {X 24.328,Y 288.978,Z 177.054,A -94.812,B 90.000,C 0.000} C_DIS
LIN {X 24.484,Y 288.965,Z 178.229,A -94.843,B 90.000,C 0.000} C_DIS
LIN {X 24.503,Y 288.963,Z 179.412,A -94.847,B 90.000,C 0.000} C_DIS
LIN {X 24.385,Y 288.973,Z 180.569,A -94.823,B 90.000,C 0.000} C_DIS
LIN {X 24.109,Y 288.996,Z 181.716,A -94.769,B 90.000,C 0.000} C_DIS
LIN {X 23.716,Y 289.029,Z 182.513,A -94.691,B 90.000,C 0.000} C_DIS
LIN {X 23.194,Y 289.071,Z 182.979,A -94.587,B 90.000,C 0.000} C_DIS
LIN {X 22.531,Y 289.123,Z 183.128,A -94.456,B 90.000,C 0.000} C_DIS
LIN {X 22.034,Y 289.162,Z 183.063,A -94.357,B 90.000,C 0.000} C_DIS
LIN {X 21.542,Y 289.199,Z 182.853,A -94.260,B 90.000,C 0.000} C_DIS
LIN {X 21.014,Y 289.238,Z 182.475,A -94.155,B 90.000,C 0.000} C_DIS
LIN {X 19.182,Y 289.362,Z 180.779,A -93.793,B 90.000,C 0.000} C_DIS
LIN {X 17.998,Y 289.441,Z 179.690,A -93.558,B 90.000,C 0.000} C_DIS
LIN {X 17.593,Y 289.466,Z 179.602,A -93.478,B 90.000,C 0.000} C_DIS
LIN {X 17.394,Y 289.478,Z 179.623,A -93.439,B 90.000,C 0.000} C_DIS
LIN {X 17.396,Y 289.478,Z 179.759,A -93.439,B 90.000,C 0.000} C_DIS
LIN {X 17.793,Y 289.454,Z 180.648,A -93.518,B 90.000,C 0.000} C_DIS
LIN {X 19.143,Y 289.367,Z 182.750,A -93.785,B 90.000,C 0.000} C_DIS
LIN {X 20.654,Y 289.264,Z 184.739,A -94.084,B 90.000,C 0.000} C_DIS
LIN {X 22.366,Y 289.135,Z 186.556,A -94.423,B 90.000,C 0.000} C_DIS
LIN {X 24.185,Y 288.989,Z 188.264,A -94.784,B 90.000,C 0.000} C_DIS
LIN {X 26.115,Y 288.819,Z 189.844,A -95.167,B 90.000,C 0.000} C_DIS
LIN {X 28.127,Y 288.630,Z 191.315,A -95.566,B 90.000,C 0.000} C_DIS
LIN {X 30.213,Y 288.419,Z 192.677,A -95.980,B 90.000,C 0.000} C_DIS
LIN {X 32.365,Y 288.188,Z 193.929,A -96.408,B 90.000,C 0.000} C_DIS
LIN {X 34.595,Y 287.927,Z 195.029,A -96.851,B 90.000,C 0.000} C_DIS
LIN {X 36.878,Y 287.642,Z 196.007,A -97.306,B 90.000,C 0.000} C_DIS
LIN {X 39.206,Y 287.334,Z 196.863,A -97.770,B 90.000,C 0.000} C_DIS
LIN {X 41.575,Y 287.002,Z 197.591,A -98.242,B 90.000,C 0.000} C_DIS
LIN {X 43.981,Y 286.645,Z 198.167,A -98.723,B 90.000,C 0.000} C_DIS
LIN {X 46.417,Y 286.260,Z 198.578,A -99.210,B 90.000,C 0.000} C_DIS
LIN {X 48.870,Y 285.848,Z 198.826,A -99.702,B 90.000,C 0.000} C_DIS
LIN {X 51.328,Y 285.416,Z 198.966,A -100.195,B 90.000,C 0.000} C_DIS
LIN {X 53.786,Y 284.960,Z 198.997,A -100.689,B 90.000,C 0.000} C_DIS
LIN {X 56.240,Y 284.489,Z 198.950,A -101.183,B 90.000,C 0.000} C_DIS
LIN {X 58.687,Y 283.997,Z 198.797,A -101.676,B 90.000,C 0.000} C_DIS
LIN {X 61.125,Y 283.482,Z 198.595,A -102.168,B 90.000,C 0.000} C_DIS
LIN {X 63.552,Y 282.947,Z 198.324,A -102.659,B 90.000,C 0.000} C_DIS
LIN {X 65.963,Y 282.395,Z 197.963,A -103.148,B 90.000,C 0.000} C_DIS
LIN {X 68.354,Y 281.827,Z 197.508,A -103.633,B 90.000,C 0.000} C_DIS
LIN {X 70.720,Y 281.243,Z 196.947,A -104.115,B 90.000,C 0.000} C_DIS
LIN {X 73.050,Y 280.647,Z 196.267,A -104.590,B 90.000,C 0.000} C_DIS
LIN {X 74.428,Y 280.287,Z 195.811,A -104.871,B 90.000,C 0.000} C_DIS
LIN {X 73.914,Y 278.354,Z 195.811,A -104.871,B 90.000,C 0.000} C_DIS
WAIT SEC 0.1
RET=EKI_SetBool("oxy","torchState",FALSE)
RET = EKI_Send("oxy","torchState")
LIN {X 69.295,Y 260.956,Z 195.811,A -104.871,B 90.000,C 0.000} C_DIS
LIN {X 20.986,Y 269.183,Z 175.483,A -94.458,B 90.000,C 0.000} C_DIS
LIN {X 22.385,Y 287.129,Z 175.483,A -94.458,B 90.000,C 0.000} C_DIS
LIN {X 22.541,Y 289.123,Z 175.483,A -94.458,B 90.000,C 0.000} C_DIS
WAIT SEC 1
RET=EKI_SetBool("oxy","torchState",TRUE)
RET = EKI_Send("oxy","torchState")
LIN {X 22.392,Y 289.134,Z 175.779,A -94.428,B 90.000,C 0.000} C_DIS
LIN {X 22.226,Y 289.147,Z 175.906,A -94.396,B 90.000,C 0.000} C_DIS
LIN {X 21.929,Y 289.170,Z 175.929,A -94.337,B 90.000,C 0.000} C_DIS
LIN {X 21.255,Y 289.220,Z 175.755,A -94.203,B 90.000,C 0.000} C_DIS
LIN {X 19.344,Y 289.354,Z 174.424,A -93.825,B 90.000,C 0.000} C_DIS
LIN {X 18.762,Y 289.392,Z 174.171,A -93.709,B 90.000,C 0.000} C_DIS
LIN {X 18.181,Y 289.430,Z 174.077,A -93.594,B 90.000,C 0.000} C_DIS
LIN {X 17.774,Y 289.455,Z 174.172,A -93.514,B 90.000,C 0.000} C_DIS
LIN {X 17.491,Y 289.472,Z 174.487,A -93.458,B 90.000,C 0.000} C_DIS
LIN {X 17.073,Y 289.497,Z 175.630,A -93.375,B 90.000,C 0.000} C_DIS
LIN {X 16.858,Y 289.510,Z 175.875,A -93.332,B 90.000,C 0.000} C_DIS
LIN {X 16.565,Y 289.527,Z 175.869,A -93.274,B 90.000,C 0.000} C_DIS
LIN {X 16.304,Y 289.541,Z 175.716,A -93.223,B 90.000,C 0.000} C_DIS
LIN {X 15.925,Y 289.562,Z 174.969,A -93.148,B 90.000,C 0.000} C_DIS
LIN {X 15.720,Y 289.574,Z 173.906,A -93.107,B 90.000,C 0.000} C_DIS
LIN {X 15.714,Y 289.574,Z 172.799,A -93.106,B 90.000,C 0.000} C_DIS
LIN {X 15.935,Y 289.562,Z 171.921,A -93.150,B 90.000,C 0.000} C_DIS
LIN {X 16.314,Y 289.541,Z 171.464,A -93.225,B 90.000,C 0.000} C_DIS
LIN {X 16.848,Y 289.510,Z 171.183,A -93.331,B 90.000,C 0.000} C_DIS
LIN {X 17.555,Y 289.468,Z 171.100,A -93.470,B 90.000,C 0.000} C_DIS
LIN {X 18.335,Y 289.420,Z 171.130,A -93.625,B 90.000,C 0.000} C_DIS
LIN {X 19.490,Y 289.344,Z 171.474,A -93.854,B 90.000,C 0.000} C_DIS
LIN {X 20.570,Y 289.270,Z 172.111,A -94.067,B 90.000,C 0.000} C_DIS
LIN {X 21.499,Y 289.202,Z 172.987,A -94.251,B 90.000,C 0.000} C_DIS
LIN {X 22.202,Y 289.149,Z 174.043,A -94.391,B 90.000,C 0.000} C_DIS
LIN {X 22.446,Y 289.130,Z 174.614,A -94.439,B 90.000,C 0.000} C_DIS
LIN {X 22.559,Y 289.121,Z 175.094,A -94.462,B 90.000,C 0.000} C_DIS
LIN {X 22.541,Y 289.123,Z 175.483,A -94.458,B 90.000,C 0.000} C_DIS
LIN {X 22.385,Y 287.129,Z 175.483,A -94.458,B 90.000,C 0.000} C_DIS
WAIT SEC 0.1
RET=EKI_SetBool("oxy","torchState",FALSE)
RET = EKI_Send("oxy","torchState")
LIN {X 20.986,Y 269.183,Z 175.483,A -94.458,B 90.000,C 0.000} C_DIS
LIN {X -126.011,Y 238.791,Z 149.638,A -62.179,B 90.000,C 0.000} C_DIS
LIN {X -134.411,Y 254.711,Z 149.638,A -62.179,B 90.000,C 0.000} C_DIS
LIN {X -135.345,Y 256.480,Z 149.638,A -62.179,B 90.000,C 0.000} C_DIS
WAIT SEC 1
RET=EKI_SetBool("oxy","torchState",TRUE)
RET = EKI_Send("oxy","torchState")
LIN {X -135.381,Y 256.461,Z 149.880,A -62.171,B 90.000,C 0.000} C_DIS
LIN {X -135.443,Y 256.428,Z 149.939,A -62.157,B 90.000,C 0.000} C_DIS
LIN {X -137.647,Y 255.250,Z 150.009,A -61.664,B 90.000,C 0.000} C_DIS
LIN {X -138.713,Y 254.674,Z 150.037,A -61.424,B 90.000,C 0.000} C_DIS
LIN {X -138.794,Y 254.630,Z 152.535,A -61.406,B 90.000,C 0.000} C_DIS
LIN {X -138.782,Y 254.636,Z 155.035,A -61.409,B 90.000,C 0.000} C_DIS
LIN {X -138.771,Y 254.642,Z 156.731,A -61.411,B 90.000,C 0.000} C_DIS
LIN {X -138.818,Y 254.616,Z 157.210,A -61.401,B 90.000,C 0.000} C_DIS
LIN {X -138.914,Y 254.564,Z 157.466,A -61.379,B 90.000,C 0.000} C_DIS
LIN {X -139.086,Y 254.470,Z 157.644,A -61.340,B 90.000,C 0.000} C_DIS
LIN {X -139.415,Y 254.290,Z 157.739,A -61.266,B 90.000,C 0.000} C_DIS
LIN {X -141.602,Y 253.078,Z 157.702,A -60.772,B 90.000,C 0.000} C_DIS
LIN {X -141.909,Y 252.907,Z 157.688,A -60.703,B 90.000,C 0.000} C_DIS
LIN {X -141.951,Y 252.883,Z 155.188,A -60.693,B 90.000,C 0.000} C_DIS
LIN {X -141.972,Y 252.871,Z 152.688,A -60.688,B 90.000,C 0.000} C_DIS
LIN {X -141.993,Y 252.860,Z 150.189,A -60.684,B 90.000,C 0.000} C_DIS
LIN {X -142.014,Y 252.848,Z 147.689,A -60.679,B 90.000,C 0.000} C_DIS
LIN {X -142.021,Y 252.844,Z 145.189,A -60.677,B 90.000,C 0.000} C_DIS
LIN {X -142.018,Y 252.845,Z 142.689,A -60.678,B 90.000,C 0.000} C_DIS
LIN {X -142.016,Y 252.846,Z 140.189,A -60.678,B 90.000,C 0.000} C_DIS
LIN {X -142.014,Y 252.848,Z 137.689,A -60.679,B 90.000,C 0.000} C_DIS
LIN {X -141.997,Y 252.857,Z 135.472,A -60.683,B 90.000,C 0.000} C_DIS
LIN {X -142.151,Y 252.771,Z 134.802,A -60.648,B 90.000,C 0.000} C_DIS
LIN {X -143.791,Y 251.836,Z 133.162,A -60.275,B 90.000,C 0.000} C_DIS
LIN {X -145.457,Y 250.877,Z 131.565,A -59.895,B 90.000,C 0.000} C_DIS
LIN {X -147.059,Y 249.947,Z 129.885,A -59.529,B 90.000,C 0.000} C_DIS
LIN {X -147.137,Y 249.901,Z 129.795,A -59.511,B 90.000,C 0.000} C_DIS
LIN {X -147.209,Y 249.859,Z 129.303,A -59.495,B 90.000,C 0.000} C_DIS
LIN {X -147.278,Y 249.818,Z 126.805,A -59.479,B 90.000,C 0.000} C_DIS
LIN {X -147.353,Y 249.774,Z 124.306,A -59.462,B 90.000,C 0.000} C_DIS
LIN {X -147.448,Y 249.718,Z 121.809,A -59.440,B 90.000,C 0.000} C_DIS
LIN {X -147.544,Y 249.661,Z 119.311,A -59.418,B 90.000,C 0.000} C_DIS
LIN {X -147.639,Y 249.605,Z 116.814,A -59.396,B 90.000,C 0.000} C_DIS
LIN {X -147.714,Y 249.561,Z 114.315,A -59.379,B 90.000,C 0.000} C_DIS
LIN {X -147.724,Y 249.555,Z 111.939,A -59.377,B 90.000,C 0.000} C_DIS
LIN {X -147.665,Y 249.590,Z 111.756,A -59.390,B 90.000,C 0.000} C_DIS
LIN {X -147.510,Y 249.681,Z 111.571,A -59.426,B 90.000,C 0.000} C_DIS
LIN {X -147.084,Y 249.932,Z 111.422,A -59.523,B 90.000,C 0.000} C_DIS
LIN {X -144.944,Y 251.175,Z 111.069,A -60.012,B 90.000,C 0.000} C_DIS
LIN {X -142.794,Y 252.402,Z 110.720,A -60.501,B 90.000,C 0.000} C_DIS
LIN {X -140.634,Y 253.617,Z 110.391,A -60.991,B 90.000,C 0.000} C_DIS
LIN {X -140.047,Y 253.943,Z 110.319,A -61.124,B 90.000,C 0.000} C_DIS
LIN {X -139.397,Y 254.300,Z 110.366,A -61.270,B 90.000,C 0.000} C_DIS
LIN {X -139.204,Y 254.406,Z 110.718,A -61.314,B 90.000,C 0.000} C_DIS
LIN {X -139.116,Y 254.454,Z 113.216,A -61.334,B 90.000,C 0.000} C_DIS
LIN {X -139.091,Y 254.467,Z 115.716,A -61.339,B 90.000,C 0.000} C_DIS
LIN {X -139.066,Y 254.481,Z 118.215,A -61.345,B 90.000,C 0.000} C_DIS
LIN {X -139.041,Y 254.495,Z 120.715,A -61.350,B 90.000,C 0.000} C_DIS
LIN {X -139.017,Y 254.508,Z 123.215,A -61.356,B 90.000,C 0.000} C_DIS
LIN {X -138.994,Y 254.520,Z 125.715,A -61.361,B 90.000,C 0.000} C_DIS
LIN {X -138.971,Y 254.533,Z 128.214,A -61.366,B 90.000,C 0.000} C_DIS
LIN {X -138.948,Y 254.546,Z 130.714,A -61.371,B 90.000,C 0.000} C_DIS
LIN {X -138.925,Y 254.558,Z 133.214,A -61.377,B 90.000,C 0.000} C_DIS
LIN {X -138.901,Y 254.571,Z 135.714,A -61.382,B 90.000,C 0.000} C_DIS
LIN {X -138.877,Y 254.584,Z 138.214,A -61.387,B 90.000,C 0.000} C_DIS
LIN {X -138.853,Y 254.598,Z 140.713,A -61.393,B 90.000,C 0.000} C_DIS
LIN {X -138.849,Y 254.600,Z 141.099,A -61.394,B 90.000,C 0.000} C_DIS
LIN {X -138.805,Y 254.624,Z 141.529,A -61.404,B 90.000,C 0.000} C_DIS
LIN {X -138.689,Y 254.687,Z 141.638,A -61.430,B 90.000,C 0.000} C_DIS
LIN {X -136.488,Y 255.872,Z 141.694,A -61.924,B 90.000,C 0.000} C_DIS
LIN {X -135.336,Y 256.484,Z 141.715,A -62.181,B 90.000,C 0.000} C_DIS
LIN {X -135.299,Y 256.504,Z 144.215,A -62.190,B 90.000,C 0.000} C_DIS
LIN {X -135.299,Y 256.504,Z 146.714,A -62.190,B 90.000,C 0.000} C_DIS
LIN {X -135.334,Y 256.485,Z 149.214,A -62.182,B 90.000,C 0.000} C_DIS
LIN {X -135.345,Y 256.480,Z 149.638,A -62.179,B 90.000,C 0.000} C_DIS
LIN {X -134.411,Y 254.711,Z 149.638,A -62.179,B 90.000,C 0.000} C_DIS
WAIT SEC 0.1
RET=EKI_SetBool("oxy","torchState",FALSE)
RET = EKI_Send("oxy","torchState")
LIN {X -126.011,Y 238.791,Z 149.638,A -62.179,B 90.000,C 0.000} C_DIS
LIN {X -138.302,Y 231.889,Z 151.587,A -59.188,B 90.000,C 0.000} C_DIS
LIN {X -147.522,Y 247.348,Z 151.587,A -59.188,B 90.000,C 0.000} C_DIS
LIN {X -148.547,Y 249.066,Z 151.587,A -59.188,B 90.000,C 0.000} C_DIS
WAIT SEC 1
RET=EKI_SetBool("oxy","torchState",TRUE)
RET = EKI_Send("oxy","torchState")
LIN {X -148.689,Y 248.981,Z 151.889,A -59.155,B 90.000,C 0.000} C_DIS
LIN {X -148.929,Y 248.838,Z 152.271,A -59.100,B 90.000,C 0.000} C_DIS
LIN {X -149.265,Y 248.636,Z 152.563,A -59.022,B 90.000,C 0.000} C_DIS
LIN {X -149.728,Y 248.358,Z 152.786,A -58.915,B 90.000,C 0.000} C_DIS
LIN {X -150.346,Y 247.984,Z 152.960,A -58.773,B 90.000,C 0.000} C_DIS
LIN {X -152.477,Y 246.678,Z 153.045,A -58.279,B 90.000,C 0.000} C_DIS
LIN {X -154.597,Y 245.353,Z 153.054,A -57.785,B 90.000,C 0.000} C_DIS
LIN {X -156.705,Y 244.010,Z 153.063,A -57.291,B 90.000,C 0.000} C_DIS
LIN {X -158.803,Y 242.650,Z 153.072,A -56.797,B 90.000,C 0.000} C_DIS
LIN {X -160.890,Y 241.275,Z 153.080,A -56.303,B 90.000,C 0.000} C_DIS
LIN {X -162.964,Y 239.879,Z 153.076,A -55.809,B 90.000,C 0.000} C_DIS
LIN {X -165.026,Y 238.466,Z 153.073,A -55.315,B 90.000,C 0.000} C_DIS
LIN {X -167.076,Y 237.035,Z 153.070,A -54.822,B 90.000,C 0.000} C_DIS
LIN {X -169.113,Y 235.586,Z 153.067,A -54.328,B 90.000,C 0.000} C_DIS
LIN {X -171.137,Y 234.119,Z 153.064,A -53.834,B 90.000,C 0.000} C_DIS
LIN {X -173.149,Y 232.634,Z 153.061,A -53.340,B 90.000,C 0.000} C_DIS
LIN {X -175.148,Y 231.133,Z 153.058,A -52.846,B 90.000,C 0.000} C_DIS
LIN {X -177.134,Y 229.614,Z 153.055,A -52.352,B 90.000,C 0.000} C_DIS
LIN {X -179.106,Y 228.079,Z 153.052,A -51.858,B 90.000,C 0.000} C_DIS
LIN {X -181.066,Y 226.526,Z 153.049,A -51.364,B 90.000,C 0.000} C_DIS
LIN {X -183.011,Y 224.956,Z 153.046,A -50.870,B 90.000,C 0.000} C_DIS
LIN {X -184.944,Y 223.370,Z 153.042,A -50.376,B 90.000,C 0.000} C_DIS
LIN {X -186.862,Y 221.768,Z 153.039,A -49.882,B 90.000,C 0.000} C_DIS
LIN {X -188.767,Y 220.149,Z 153.036,A -49.388,B 90.000,C 0.000} C_DIS
LIN {X -190.658,Y 218.513,Z 153.023,A -48.895,B 90.000,C 0.000} C_DIS
LIN {X -192.534,Y 216.861,Z 153.004,A -48.401,B 90.000,C 0.000} C_DIS
LIN {X -194.396,Y 215.194,Z 152.984,A -47.907,B 90.000,C 0.000} C_DIS
LIN {X -196.244,Y 213.510,Z 152.964,A -47.413,B 90.000,C 0.000} C_DIS
LIN {X -198.078,Y 211.811,Z 152.944,A -46.919,B 90.000,C 0.000} C_DIS
LIN {X -199.896,Y 210.095,Z 152.926,A -46.425,B 90.000,C 0.000} C_DIS
LIN {X -201.701,Y 208.366,Z 152.911,A -45.931,B 90.000,C 0.000} C_DIS
LIN {X -203.489,Y 206.618,Z 152.896,A -45.437,B 90.000,C 0.000} C_DIS
